// TIA Portal V20 export
FUNCTION_BLOCK "LSicar_KistlerPress"   // FB2, LAD
{ S7_Optimized_Access := 'TRUE' }
VERSION : 0.1
// stored: AutoNumber true, IsIECCheckEnabled false, IsRetainMemResEnabled false, MemoryReserve 100, SetENOAutomatically false, UDAEnableTagReadback false
   VAR_INPUT
      plantidentifier { ExternalAccessible := 'False'; ExternalVisible := 'False'; ExternalWritable := 'False'} : WString[24];
      CarrierID { ExternalAccessible := 'False'; ExternalVisible := 'False'; ExternalWritable := 'False'} : WString[9];
      mpSerialNumber { ExternalAccessible := 'False'; ExternalVisible := 'False'; ExternalWritable := 'False'} : String[24];
      additionaAlarmText { ExternalAccessible := 'False'; ExternalVisible := 'False'; ExternalWritable := 'False'} : WString[15];
      tecUnitNumber { ExternalAccessible := 'False'; ExternalVisible := 'False'; ExternalWritable := 'False'} : Int;
      enableBlock { ExternalAccessible := 'False'; ExternalVisible := 'False'; ExternalWritable := 'False'} : Bool := TRUE;
      HardwareOK { ExternalAccessible := 'False'; ExternalVisible := 'False'; ExternalWritable := 'False'} : Bool := TRUE;
      SafetyOK { ExternalAccessible := 'False'; ExternalVisible := 'False'; ExternalWritable := 'False'} : Bool := TRUE;
      servoNotInstalled { ExternalAccessible := 'False'; ExternalVisible := 'False'; ExternalWritable := 'False'} : Bool;
      hardwareID1 { ExternalAccessible := 'False'; ExternalVisible := 'False'; ExternalWritable := 'False'} : HW_IO;
      hardwareID2 { ExternalAccessible := 'False'; ExternalVisible := 'False'; ExternalWritable := 'False'} : HW_IO;
      smartClientIPAddress { ExternalAccessible := 'False'; ExternalVisible := 'False'; ExternalWritable := 'False'} : String[20];
      mpNumber { ExternalAccessible := 'False'; ExternalVisible := 'False'; ExternalWritable := 'False'} : Byte;
      cfgAdd { ExternalAccessible := 'False'; ExternalVisible := 'False'; ExternalWritable := 'False'} : Byte;
      CfgLentgh { ExternalAccessible := 'False'; ExternalVisible := 'False'; ExternalWritable := 'False'} : Byte;
      SelectPageNumber { ExternalAccessible := 'False'; ExternalVisible := 'False'; ExternalWritable := 'False'} : Byte;
      selectSequence { ExternalAccessible := 'False'; ExternalVisible := 'False'; ExternalWritable := 'False'} : Byte;
      extStopRequest { ExternalAccessible := 'False'; ExternalVisible := 'False'; ExternalWritable := 'False'} : Bool;
      strobeEnable { ExternalAccessible := 'False'; ExternalVisible := 'False'; ExternalWritable := 'False'} : Bool;
      startTL { ExternalAccessible := 'False'; ExternalVisible := 'False'; ExternalWritable := 'False'} : Bool;
      autoRunSequence { ExternalAccessible := 'False'; ExternalVisible := 'False'; ExternalWritable := 'False'} : Bool := FALSE;
      autoHomePosition { ExternalAccessible := 'False'; ExternalVisible := 'False'; ExternalWritable := 'False'} : Bool;
      autoDriveToReferencePosition { ExternalAccessible := 'False'; ExternalVisible := 'False'; ExternalWritable := 'False'} : Bool;
      JogFwd { ExternalAccessible := 'False'; ExternalVisible := 'False'; ExternalWritable := 'False'} : Bool;
      JogNeq { ExternalAccessible := 'False'; ExternalVisible := 'False'; ExternalWritable := 'False'} : Bool;
      continuewait { ExternalAccessible := 'False'; ExternalVisible := 'False'; ExternalWritable := 'False'} : Bool;
      SequenceEndReset { ExternalAccessible := 'False'; ExternalVisible := 'False'; ExternalWritable := 'False'} : Bool;
      enableRunSequence { ExternalAccessible := 'False'; ExternalVisible := 'False'; ExternalWritable := 'False'} : Bool := TRUE;
      enablehomePos { ExternalAccessible := 'False'; ExternalVisible := 'False'; ExternalWritable := 'False'} : Bool := TRUE;
      externalAlarm { ExternalAccessible := 'False'; ExternalVisible := 'False'; ExternalWritable := 'False'} : Bool;
      runWithoutEnable { ExternalAccessible := 'False'; ExternalVisible := 'False'; ExternalWritable := 'False'} : Bool;
      hideAlarmAll { ExternalAccessible := 'False'; ExternalVisible := 'False'; ExternalWritable := 'False'} : Bool;
      hideAlarmMask { ExternalAccessible := 'False'; ExternalVisible := 'False'; ExternalWritable := 'False'} : DWord;
      OpModeUserInterfaceOut { ExternalAccessible := 'False'; ExternalVisible := 'False'; ExternalWritable := 'False'} : "LSicar_typeOpmodeOut";
      timeOperation { ExternalAccessible := 'False'; ExternalVisible := 'False'; ExternalWritable := 'False'} : Time;
      timeExtStop { ExternalAccessible := 'False'; ExternalVisible := 'False'; ExternalWritable := 'False'} : Time;
      parameters { ExternalAccessible := 'False'; ExternalVisible := 'False'; ExternalWritable := 'False'} : "LDrive_typeKistlerParameters";
   END_VAR
   VAR_OUTPUT
      GeneralAlarm { ExternalAccessible := 'False'; ExternalVisible := 'False'; ExternalWritable := 'False'} : Bool;
      AutomaticActive { ExternalAccessible := 'False'; ExternalVisible := 'False'; ExternalWritable := 'False'} : Bool;
      okTotal { ExternalAccessible := 'False'; ExternalVisible := 'False'; ExternalWritable := 'False'} : Bool;
      nokTotal { ExternalAccessible := 'False'; ExternalVisible := 'False'; ExternalWritable := 'False'} : Bool;
      noPass { ExternalAccessible := 'False'; ExternalVisible := 'False'; ExternalWritable := 'False'} : Bool;
      sequenceRunning { ExternalAccessible := 'False'; ExternalVisible := 'False'; ExternalWritable := 'False'} : Bool;
      sequenceStopped { ExternalAccessible := 'False'; ExternalVisible := 'False'; ExternalWritable := 'False'} : Bool;
      Sequenceend { ExternalAccessible := 'False'; ExternalVisible := 'False'; ExternalWritable := 'False'} : Bool;
      homePos { ExternalAccessible := 'False'; ExternalVisible := 'False'; ExternalWritable := 'False'} : Bool;
      referencePos { ExternalAccessible := 'False'; ExternalVisible := 'False'; ExternalWritable := 'False'} : Bool;
      waitContinue { ExternalAccessible := 'False'; ExternalVisible := 'False'; ExternalWritable := 'False'} : Bool;
      ready { ExternalAccessible := 'False'; ExternalVisible := 'False'; ExternalWritable := 'False'} : Bool;
      pvCurrentValueX { ExternalAccessible := 'False'; ExternalVisible := 'False'; ExternalWritable := 'False'} : Real;
      pvCurrentValueY { ExternalAccessible := 'False'; ExternalVisible := 'False'; ExternalWritable := 'False'} : Real;
      pvCurveXminX { ExternalAccessible := 'False'; ExternalVisible := 'False'; ExternalWritable := 'False'} : Real;
      pvCurveXmaxX { ExternalAccessible := 'False'; ExternalVisible := 'False'; ExternalWritable := 'False'} : Real;
      pvCurveYminY { ExternalAccessible := 'False'; ExternalVisible := 'False'; ExternalWritable := 'False'} : Real;
      pvCurveYmaxY { ExternalAccessible := 'False'; ExternalVisible := 'False'; ExternalWritable := 'False'} : Real;
      customeProcessValues { ExternalAccessible := 'False'; ExternalVisible := 'False'; ExternalWritable := 'False'} : "LDrive_typeKistlerProcessValues";
      displayeservoJogSpeed { ExternalAccessible := 'False'; ExternalVisible := 'False'; ExternalWritable := 'False'} : Real;
      standstill { ExternalAccessible := 'False'; ExternalVisible := 'False'; ExternalWritable := 'False'} : Bool;
      MeasurementProgramEcho { ExternalAccessible := 'False'; ExternalVisible := 'False'; ExternalWritable := 'False'} : DInt;
      currentLabel { ExternalAccessible := 'False'; ExternalVisible := 'False'; ExternalWritable := 'False'} : Byte;
   END_VAR
   VAR_IN_OUT
      interfaceHmi : Array[*] of "LDrive_typeKistlerHmi";
   END_VAR
   VAR
      statDataExchangeReceive { ExternalAccessible := 'False'; ExternalVisible := 'False'; ExternalWritable := 'False'} : "LDrive_typeKistlerPressDataRecv";
      statDataExchangeSend { ExternalAccessible := 'False'; ExternalVisible := 'False'; ExternalWritable := 'False'} : "LDrive_typeKistlerPressDataSend";
      statInstruction { ExternalAccessible := 'False'; ExternalVisible := 'False'; ExternalWritable := 'False'} : Struct
         timeroperation { ExternalAccessible := 'False'; ExternalVisible := 'False'; ExternalWritable := 'False'; S7_SetPoint := 'True'} : IEC_TIMER;
         driveEnableTMR { ExternalAccessible := 'False'; ExternalVisible := 'False'; ExternalWritable := 'False'; S7_SetPoint := 'True'} : IEC_TIMER;
      END_STRUCT;
      stateAlarm { ExternalAccessible := 'False'; ExternalVisible := 'False'; ExternalWritable := 'False'} : Struct
         spare0 { ExternalAccessible := 'False'; ExternalVisible := 'False'; ExternalWritable := 'False'} : Bool;
         hardwareNOK { ExternalAccessible := 'False'; ExternalVisible := 'False'; ExternalWritable := 'False'} : Bool;
         driveenabledNOK { ExternalAccessible := 'False'; ExternalVisible := 'False'; ExternalWritable := 'False'} : Bool;
         enableRunSequence { ExternalAccessible := 'False'; ExternalVisible := 'False'; ExternalWritable := 'False'} : Bool;
         enableHomePos { ExternalAccessible := 'False'; ExternalVisible := 'False'; ExternalWritable := 'False'} : Bool;
         timerMonitorRunSequence { ExternalAccessible := 'False'; ExternalVisible := 'False'; ExternalWritable := 'False'} : Bool;
         timerMonitorHomePos { ExternalAccessible := 'False'; ExternalVisible := 'False'; ExternalWritable := 'False'} : Bool;
         timerMonitorReferencePos { ExternalAccessible := 'False'; ExternalVisible := 'False'; ExternalWritable := 'False'} : Bool;
         noContinueWaitCommand { ExternalAccessible := 'False'; ExternalVisible := 'False'; ExternalWritable := 'False'} : Bool;
         alarm { ExternalAccessible := 'False'; ExternalVisible := 'False'; ExternalWritable := 'False'} : Bool;
         spare11 { ExternalAccessible := 'False'; ExternalVisible := 'False'; ExternalWritable := 'False'} : Bool;
         smesActive { ExternalAccessible := 'False'; ExternalVisible := 'False'; ExternalWritable := 'False'} : Bool;
         safetyNOK { ExternalAccessible := 'False'; ExternalVisible := 'False'; ExternalWritable := 'False'} : Bool;
         smst2active { ExternalAccessible := 'False'; ExternalVisible := 'False'; ExternalWritable := 'False'} : Bool;
         smm1active { ExternalAccessible := 'False'; ExternalVisible := 'False'; ExternalWritable := 'False'} : Bool;
         serialnumbermismatch { ExternalAccessible := 'False'; ExternalVisible := 'False'; ExternalWritable := 'False'} : Bool;
         transmissionFault { ExternalAccessible := 'False'; ExternalVisible := 'False'; ExternalWritable := 'False'} : Bool;
         remoteControlNotActive { ExternalAccessible := 'False'; ExternalVisible := 'False'; ExternalWritable := 'False'} : Bool;
      END_STRUCT;
      stateHideAlarm { ExternalAccessible := 'False'; ExternalVisible := 'False'; ExternalWritable := 'False'} : Struct
         spare0 { ExternalAccessible := 'False'; ExternalVisible := 'False'; ExternalWritable := 'False'} : Bool;
         hardwareNOK { ExternalAccessible := 'False'; ExternalVisible := 'False'; ExternalWritable := 'False'} : Bool;
         transmissionFault { ExternalAccessible := 'False'; ExternalVisible := 'False'; ExternalWritable := 'False'} : Bool;
         driveEnabledNOK { ExternalAccessible := 'False'; ExternalVisible := 'False'; ExternalWritable := 'False'} : Bool;
         enableRunSequence { ExternalAccessible := 'False'; ExternalVisible := 'False'; ExternalWritable := 'False'} : Bool;
         enableHomePos { ExternalAccessible := 'False'; ExternalVisible := 'False'; ExternalWritable := 'False'} : Bool;
         timerMonitorRunSequence { ExternalAccessible := 'False'; ExternalVisible := 'False'; ExternalWritable := 'False'} : Bool;
         timerMonitorHomePos { ExternalAccessible := 'False'; ExternalVisible := 'False'; ExternalWritable := 'False'} : Bool;
         timerMonitorReferencePos { ExternalAccessible := 'False'; ExternalVisible := 'False'; ExternalWritable := 'False'} : Bool;
         noContinueWaitCommand { ExternalAccessible := 'False'; ExternalVisible := 'False'; ExternalWritable := 'False'} : Bool;
         Alarm { ExternalAccessible := 'False'; ExternalVisible := 'False'; ExternalWritable := 'False'} : Bool;
         spare11 { ExternalAccessible := 'False'; ExternalVisible := 'False'; ExternalWritable := 'False'} : Bool;
         smesactive { ExternalAccessible := 'False'; ExternalVisible := 'False'; ExternalWritable := 'False'} : Bool;
         safetyNOK { ExternalAccessible := 'False'; ExternalVisible := 'False'; ExternalWritable := 'False'} : Bool;
         smst2active { ExternalAccessible := 'False'; ExternalVisible := 'False'; ExternalWritable := 'False'} : Bool;
         smm1Active { ExternalAccessible := 'False'; ExternalVisible := 'False'; ExternalWritable := 'False'} : Bool;
      END_STRUCT;
      aux { ExternalAccessible := 'False'; ExternalVisible := 'False'; ExternalWritable := 'False'} : Struct
         generalAlarm { ExternalAccessible := 'False'; ExternalVisible := 'False'; ExternalWritable := 'False'} : Bool := false;
         plantIdentifier { ExternalAccessible := 'False'; ExternalVisible := 'False'; ExternalWritable := 'False'} : String[24];
         HideAlarmAll { ExternalAccessible := 'False'; ExternalVisible := 'False'; ExternalWritable := 'False'} : Bool := false;
         manualMode { ExternalAccessible := 'False'; ExternalVisible := 'False'; ExternalWritable := 'False'} : Bool := false;
         automaticMode { ExternalAccessible := 'False'; ExternalVisible := 'False'; ExternalWritable := 'False'} : Bool := false;
         singleStepMode { ExternalAccessible := 'False'; ExternalVisible := 'False'; ExternalWritable := 'False'} : Bool := false;
         setupMode { ExternalAccessible := 'False'; ExternalVisible := 'False'; ExternalWritable := 'False'} : Bool := false;
         externalAlarm { ExternalAccessible := 'False'; ExternalVisible := 'False'; ExternalWritable := 'False'} : Bool := false;
         alarmPdNoChange { ExternalAccessible := 'False'; ExternalVisible := 'False'; ExternalWritable := 'False'} : Bool := false;
         internalAlarmPdNoChange { ExternalAccessible := 'False'; ExternalVisible := 'False'; ExternalWritable := 'False'} : Bool := false;
         lastAlarmNoPD { ExternalAccessible := 'False'; ExternalVisible := 'False'; ExternalWritable := 'False'} : UInt := 0;
         lastInternalAlarmNoPD { ExternalAccessible := 'False'; ExternalVisible := 'False'; ExternalWritable := 'False'} : UInt := 0;
         enableAdvancedCodeView { ExternalAccessible := 'False'; ExternalVisible := 'False'; ExternalWritable := 'False'} : Bool := false;
         enableReverseCodeView { ExternalAccessible := 'False'; ExternalVisible := 'False'; ExternalWritable := 'False'} : Bool := false;
         codeViewAdvancedFilter { ExternalAccessible := 'False'; ExternalVisible := 'False'; ExternalWritable := 'False'} : WString[48];
         codeViewReverseFilter { ExternalAccessible := 'False'; ExternalVisible := 'False'; ExternalWritable := 'False'} : WString[48];
         iecTimer1 { ExternalAccessible := 'False'; ExternalVisible := 'False'; ExternalWritable := 'False'} : TON_TIME;
         logicEnable { ExternalAccessible := 'False'; ExternalVisible := 'False'; ExternalWritable := 'False'; S7_SetPoint := 'True'} : Bool := false;
         runSequence { ExternalAccessible := 'False'; ExternalVisible := 'False'; ExternalWritable := 'False'} : Bool := false;
         sequenceEnd { ExternalAccessible := 'False'; ExternalVisible := 'False'; ExternalWritable := 'False'} : Bool := false;
         dataStrobed { ExternalAccessible := 'False'; ExternalVisible := 'False'; ExternalWritable := 'False'} : Bool := false;
         SeqEnd { ExternalAccessible := 'False'; ExternalVisible := 'False'; ExternalWritable := 'False'} : Bool := false;
         remoteControl { ExternalAccessible := 'False'; ExternalVisible := 'False'; ExternalWritable := 'False'} : Bool := false;
         manualDataStrobe { ExternalAccessible := 'False'; ExternalVisible := 'False'; ExternalWritable := 'False'} : Bool := false;
         kistlerDataDB { ExternalAccessible := 'False'; ExternalVisible := 'False'; ExternalWritable := 'False'} : Int := 0;
         pulse { ExternalAccessible := 'False'; ExternalVisible := 'False'; ExternalWritable := 'False'} : Array[0..16] of Bool;
         Interface { ExternalAccessible := 'False'; ExternalVisible := 'False'; ExternalWritable := 'False'} : DWord;
      END_STRUCT;
      ons { ExternalAccessible := 'False'; ExternalVisible := 'False'; ExternalWritable := 'False'} : Array[0..16] of Bool;
      statTimeExpire { ExternalAccessible := 'False'; ExternalVisible := 'False'; ExternalWritable := 'False'} : Struct
         operating { ExternalAccessible := 'False'; ExternalVisible := 'False'; ExternalWritable := 'False'} : Bool;
         position_pLeft { ExternalAccessible := 'False'; ExternalVisible := 'False'; ExternalWritable := 'False'} : Bool;
         selaypair_mon { ExternalAccessible := 'False'; ExternalVisible := 'False'; ExternalWritable := 'False'} : Bool;
         dwellTimeWork { ExternalAccessible := 'False'; ExternalVisible := 'False'; ExternalWritable := 'False'} : Bool;
         dwellTimeHome { ExternalAccessible := 'False'; ExternalVisible := 'False'; ExternalWritable := 'False'} : Bool;
      END_STRUCT;
      statAlarmtextHeader { ExternalAccessible := 'False'; ExternalVisible := 'False'; ExternalWritable := 'False'} : WString[60];
      statAlarmtextFooter { ExternalAccessible := 'False'; ExternalVisible := 'False'; ExternalWritable := 'False'} : WString[24];
      statPalletID { ExternalAccessible := 'False'; ExternalVisible := 'False'; ExternalWritable := 'False'} : WString[9];
      statAlarmNoPD { ExternalAccessible := 'False'; ExternalVisible := 'False'; ExternalWritable := 'False'} : UInt;
      statInternalAlarmNoPD { ExternalAccessible := 'False'; ExternalVisible := 'False'; ExternalWritable := 'False'} : UInt;
      statHideAlarmMessagesPD { ExternalAccessible := 'False'; ExternalVisible := 'False'; ExternalWritable := 'False'} : Bool;
      statGlobalTecunitWarningTestListItem { ExternalAccessible := 'False'; ExternalVisible := 'False'; ExternalWritable := 'False'} : USInt := 92;
      statCodeViewAdvanceCond { ExternalAccessible := 'False'; ExternalVisible := 'False'; ExternalWritable := 'False'} : TON_TIME;
      statCodeViewReverseCond { ExternalAccessible := 'False'; ExternalVisible := 'False'; ExternalWritable := 'False'; S7_SetPoint := 'True'} : TON_TIME;
      statdriveDelayTimer { ExternalAccessible := 'False'; ExternalVisible := 'False'; ExternalWritable := 'False'; S7_SetPoint := 'True'} : TON_TIME;
      tof { ExternalAccessible := 'False'; ExternalVisible := 'False'; ExternalWritable := 'False'; S7_SetPoint := 'True'} : TON_TIME;
      statSerialByteIndex { ExternalAccessible := 'False'; ExternalVisible := 'False'; ExternalWritable := 'False'; S7_SetPoint := 'True'} : Int;
      statAlarmByteIndex { ExternalAccessible := 'False'; ExternalVisible := 'False'; ExternalWritable := 'False'} : Int;
      statStringIndex { ExternalAccessible := 'False'; ExternalVisible := 'False'; ExternalWritable := 'False'} : Int;
      statSerialOutput { ExternalAccessible := 'False'; ExternalVisible := 'False'; ExternalWritable := 'False'} : String[24];
      instKistlerOnDelay { ExternalAccessible := 'False'; ExternalVisible := 'False'; ExternalWritable := 'False'} : TON_TIME;
      internalFaultCode { ExternalAccessible := 'False'; ExternalVisible := 'False'; ExternalWritable := 'False'; S7_SetPoint := 'True'} : Array[0..63] of Bool;
      AlarmTextConstants { ExternalAccessible := 'False'; ExternalVisible := 'False'; ExternalWritable := 'False'} : Array[0..63] of Int;
      i { ExternalAccessible := 'False'; ExternalVisible := 'False'; ExternalWritable := 'False'} : Int;
   END_VAR
   VAR_TEMP
      tempReturnValueRead : Int;
      tempReturnValueWrite : Int;
      tempMPEcho : SInt;
      tempReadOK : Bool;
      tempWriteOK : Bool;
      tempValue : DWord;
      tempString : String[24];
      tempSerialLength : USInt;
      tempIndex : USInt;
      tempDword : DWord;
      tempErrorValue : Int;
      tempDint : DInt;
   END_VAR
   VAR CONSTANT
      cfgKistlerOnDelay : Time := T#1s;
   END_VAR
   VAR_TEMP   // added for the SCL form of the ladder/FBD networks
      _w1 : Bool;
      _w2 : Bool;
      _w3 : Bool;
      _w4 : Bool;
      _w5 : Bool;
      _w6 : Bool;
      _w7 : Bool;
   END_VAR
BEGIN

REGION Network 1 (SCL): Read RAW Data from Kistler
       #tempReturnValueRead := DPRD_DAT(LADDR := #hardwareID1, RECORD => #statDataExchangeReceive);    // Read from Kistler
END_REGION

REGION Network 2: Read OK
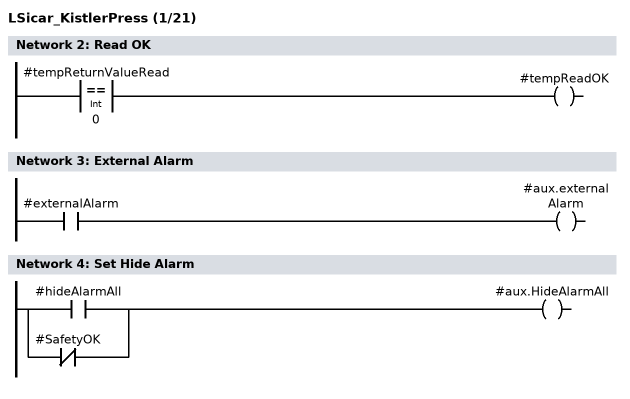
   RUNG wire#powerrail
      { S7_Templates := "SrcType := Int" } EQ_Contact(in1 := #tempReturnValueRead, in2 := 0)
      Coil( #tempReadOK )
   END_RUNG
   // the same network as SCL:
   #tempReadOK := #tempReturnValueRead = 0;
END_REGION

REGION Network 3: External Alarm
   RUNG wire#powerrail
      Contact( #externalAlarm )
      Coil( #aux.externalAlarm )
   END_RUNG
   // the same network as SCL:
   #aux.externalAlarm := #externalAlarm;
END_REGION

REGION Network 4: Set Hide Alarm
   RUNG wire#powerrail
      Contact( #hideAlarmAll )
      wire#w1
      Coil( #aux.HideAlarmAll )
   END_RUNG
   RUNG wire#powerrail
      I_Contact( #SafetyOK )
   END_RUNG wire#w1
   // the same network as SCL:
   #aux.HideAlarmAll := #hideAlarmAll OR NOT #SafetyOK;
END_REGION

REGION Network 5: Hide Alarm
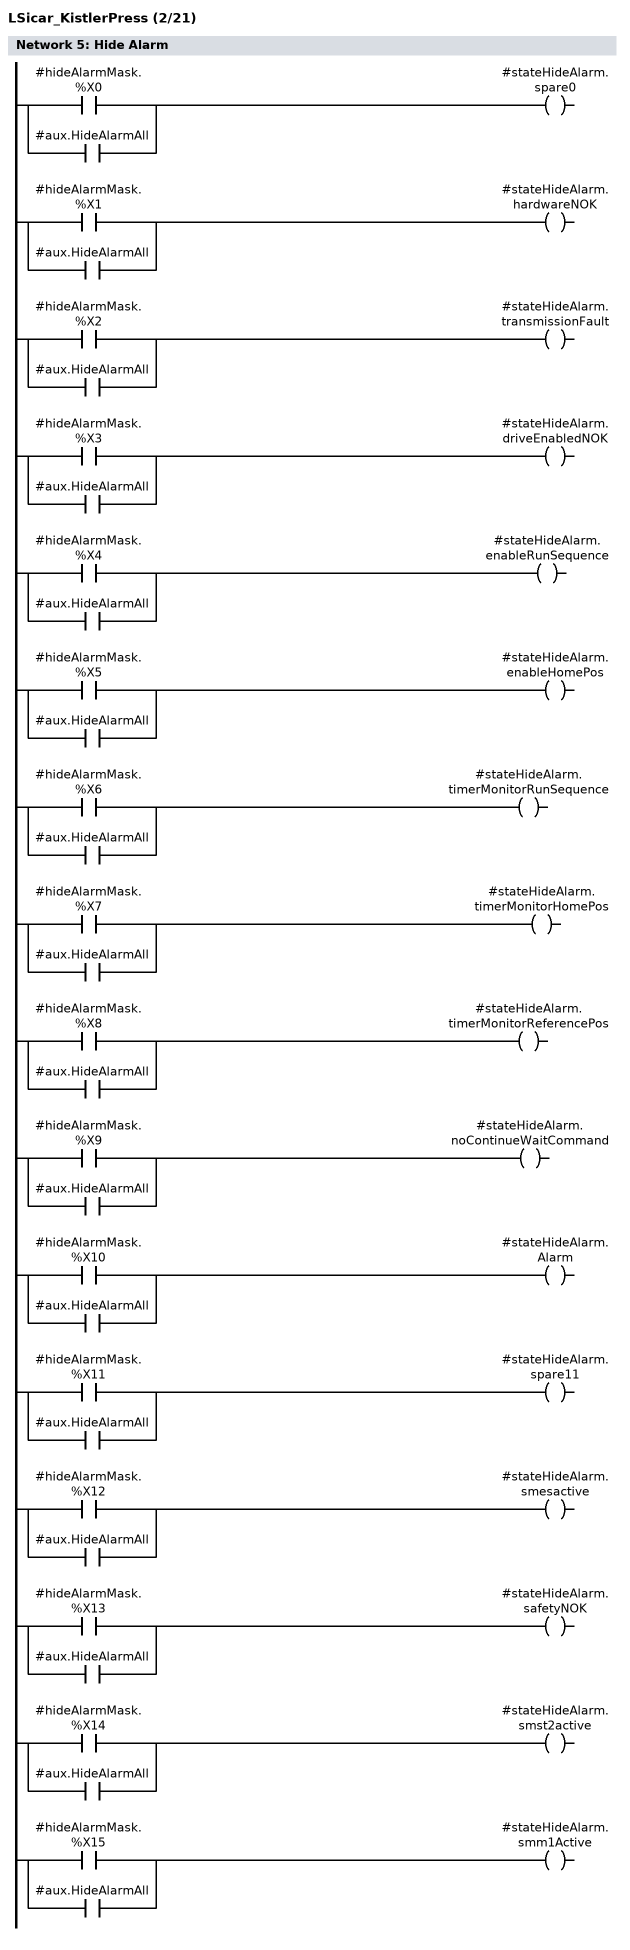
   RUNG wire#powerrail
      Contact( #hideAlarmMask.%X0 )
      wire#w1
      Coil( #stateHideAlarm.spare0 )
   END_RUNG
   RUNG wire#powerrail
      Contact( #aux.HideAlarmAll )
   END_RUNG wire#w1
   RUNG wire#powerrail
      Contact( #hideAlarmMask.%X1 )
      wire#w2
      Coil( #stateHideAlarm.hardwareNOK )
   END_RUNG
   RUNG wire#powerrail
      Contact( #aux.HideAlarmAll )
   END_RUNG wire#w2
   RUNG wire#powerrail
      Contact( #hideAlarmMask.%X2 )
      wire#w3
      Coil( #stateHideAlarm.transmissionFault )
   END_RUNG
   RUNG wire#powerrail
      Contact( #aux.HideAlarmAll )
   END_RUNG wire#w3
   RUNG wire#powerrail
      Contact( #hideAlarmMask.%X3 )
      wire#w4
      Coil( #stateHideAlarm.driveEnabledNOK )
   END_RUNG
   RUNG wire#powerrail
      Contact( #aux.HideAlarmAll )
   END_RUNG wire#w4
   RUNG wire#powerrail
      Contact( #hideAlarmMask.%X4 )
      wire#w5
      Coil( #stateHideAlarm.enableRunSequence )
   END_RUNG
   RUNG wire#powerrail
      Contact( #aux.HideAlarmAll )
   END_RUNG wire#w5
   RUNG wire#powerrail
      Contact( #hideAlarmMask.%X5 )
      wire#w6
      Coil( #stateHideAlarm.enableHomePos )
   END_RUNG
   RUNG wire#powerrail
      Contact( #aux.HideAlarmAll )
   END_RUNG wire#w6
   RUNG wire#powerrail
      Contact( #hideAlarmMask.%X6 )
      wire#w7
      Coil( #stateHideAlarm.timerMonitorRunSequence )
   END_RUNG
   RUNG wire#powerrail
      Contact( #aux.HideAlarmAll )
   END_RUNG wire#w7
   RUNG wire#powerrail
      Contact( #hideAlarmMask.%X7 )
      wire#w8
      Coil( #stateHideAlarm.timerMonitorHomePos )
   END_RUNG
   RUNG wire#powerrail
      Contact( #aux.HideAlarmAll )
   END_RUNG wire#w8
   RUNG wire#powerrail
      Contact( #hideAlarmMask.%X8 )
      wire#w9
      Coil( #stateHideAlarm.timerMonitorReferencePos )
   END_RUNG
   RUNG wire#powerrail
      Contact( #aux.HideAlarmAll )
   END_RUNG wire#w9
   RUNG wire#powerrail
      Contact( #hideAlarmMask.%X9 )
      wire#w10
      Coil( #stateHideAlarm.noContinueWaitCommand )
   END_RUNG
   RUNG wire#powerrail
      Contact( #aux.HideAlarmAll )
   END_RUNG wire#w10
   RUNG wire#powerrail
      Contact( #hideAlarmMask.%X10 )
      wire#w11
      Coil( #stateHideAlarm.Alarm )
   END_RUNG
   RUNG wire#powerrail
      Contact( #aux.HideAlarmAll )
   END_RUNG wire#w11
   RUNG wire#powerrail
      Contact( #hideAlarmMask.%X11 )
      wire#w12
      Coil( #stateHideAlarm.spare11 )
   END_RUNG
   RUNG wire#powerrail
      Contact( #aux.HideAlarmAll )
   END_RUNG wire#w12
   RUNG wire#powerrail
      Contact( #hideAlarmMask.%X12 )
      wire#w13
      Coil( #stateHideAlarm.smesactive )
   END_RUNG
   RUNG wire#powerrail
      Contact( #aux.HideAlarmAll )
   END_RUNG wire#w13
   RUNG wire#powerrail
      Contact( #hideAlarmMask.%X13 )
      wire#w14
      Coil( #stateHideAlarm.safetyNOK )
   END_RUNG
   RUNG wire#powerrail
      Contact( #aux.HideAlarmAll )
   END_RUNG wire#w14
   RUNG wire#powerrail
      Contact( #hideAlarmMask.%X14 )
      wire#w15
      Coil( #stateHideAlarm.smst2active )
   END_RUNG
   RUNG wire#powerrail
      Contact( #aux.HideAlarmAll )
   END_RUNG wire#w15
   RUNG wire#powerrail
      Contact( #hideAlarmMask.%X15 )
      wire#w16
      Coil( #stateHideAlarm.smm1Active )
   END_RUNG
   RUNG wire#powerrail
      Contact( #aux.HideAlarmAll )
   END_RUNG wire#w16
   // the same network as SCL:
   #stateHideAlarm.spare0 := #hideAlarmMask.%X0 OR #aux.HideAlarmAll;
   #stateHideAlarm.hardwareNOK := #hideAlarmMask.%X1 OR #aux.HideAlarmAll;
   #stateHideAlarm.transmissionFault := #hideAlarmMask.%X2 OR #aux.HideAlarmAll;
   #stateHideAlarm.driveEnabledNOK := #hideAlarmMask.%X3 OR #aux.HideAlarmAll;
   #stateHideAlarm.enableRunSequence := #hideAlarmMask.%X4 OR #aux.HideAlarmAll;
   #stateHideAlarm.enableHomePos := #hideAlarmMask.%X5 OR #aux.HideAlarmAll;
   #stateHideAlarm.timerMonitorRunSequence := #hideAlarmMask.%X6 OR #aux.HideAlarmAll;
   #stateHideAlarm.timerMonitorHomePos := #hideAlarmMask.%X7 OR #aux.HideAlarmAll;
   #stateHideAlarm.timerMonitorReferencePos := #hideAlarmMask.%X8 OR #aux.HideAlarmAll;
   #stateHideAlarm.noContinueWaitCommand := #hideAlarmMask.%X9 OR #aux.HideAlarmAll;
   #stateHideAlarm.Alarm := #hideAlarmMask.%X10 OR #aux.HideAlarmAll;
   #stateHideAlarm.spare11 := #hideAlarmMask.%X11 OR #aux.HideAlarmAll;
   #stateHideAlarm.smesactive := #hideAlarmMask.%X12 OR #aux.HideAlarmAll;
   #stateHideAlarm.safetyNOK := #hideAlarmMask.%X13 OR #aux.HideAlarmAll;
   #stateHideAlarm.smst2active := #hideAlarmMask.%X14 OR #aux.HideAlarmAll;
   #stateHideAlarm.smm1Active := #hideAlarmMask.%X15 OR #aux.HideAlarmAll;
END_REGION

REGION Network 6: Mode Selection
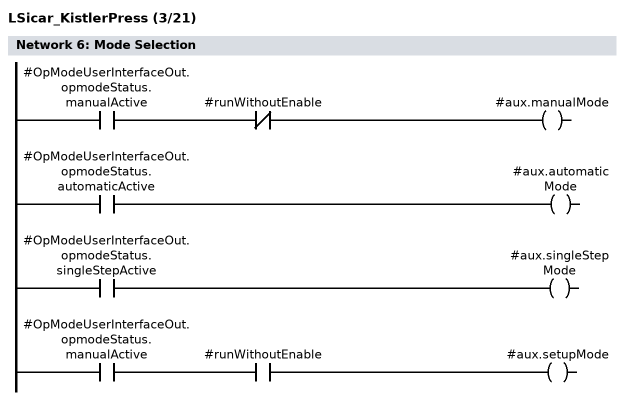
   RUNG wire#powerrail
      Contact( #OpModeUserInterfaceOut.opmodeStatus.manualActive )
      I_Contact( #runWithoutEnable )
      Coil( #aux.manualMode )
   END_RUNG
   RUNG wire#powerrail
      Contact( #OpModeUserInterfaceOut.opmodeStatus.automaticActive )
      Coil( #aux.automaticMode )
   END_RUNG
   RUNG wire#powerrail
      Contact( #OpModeUserInterfaceOut.opmodeStatus.singleStepActive )
      Coil( #aux.singleStepMode )
   END_RUNG
   RUNG wire#powerrail
      Contact( #OpModeUserInterfaceOut.opmodeStatus.manualActive )
      Contact( #runWithoutEnable )
      Coil( #aux.setupMode )
   END_RUNG
   // the same network as SCL:
   #aux.manualMode := #OpModeUserInterfaceOut.opmodeStatus.manualActive AND NOT #runWithoutEnable;
   #aux.automaticMode := #OpModeUserInterfaceOut.opmodeStatus.automaticActive;
   #aux.singleStepMode := #OpModeUserInterfaceOut.opmodeStatus.singleStepActive;
   #aux.setupMode := #OpModeUserInterfaceOut.opmodeStatus.manualActive AND #runWithoutEnable;
END_REGION

REGION Network 7: Clear Faults
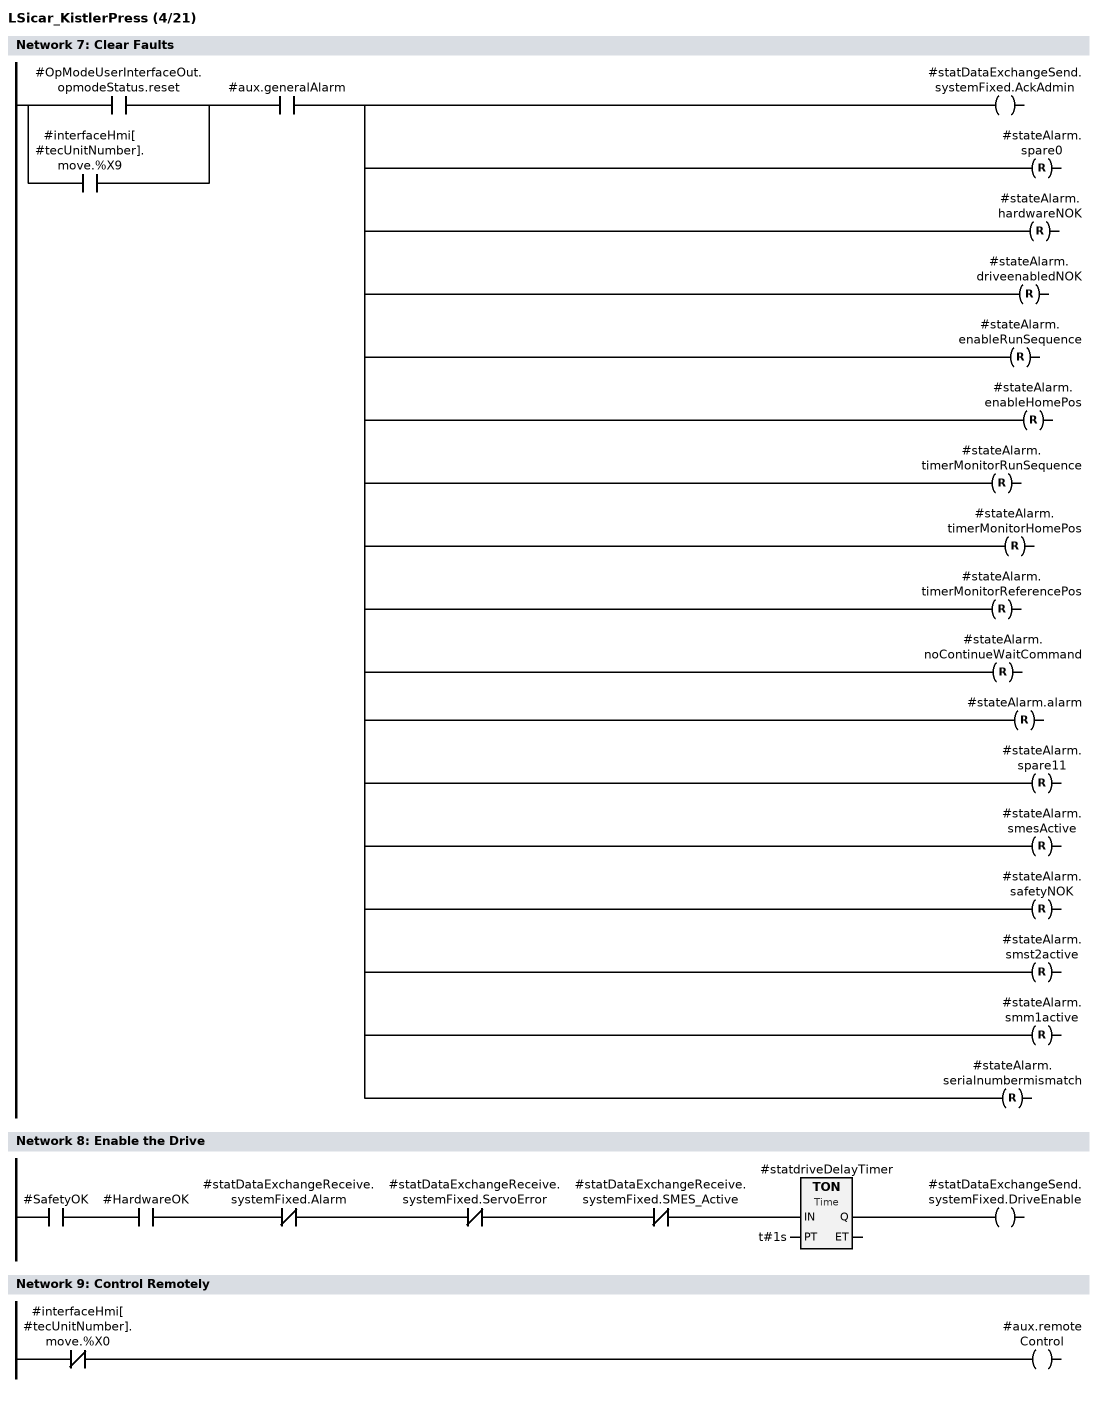
   RUNG wire#powerrail
      Contact( #OpModeUserInterfaceOut.opmodeStatus.reset )
      wire#w1
      Contact( #aux.generalAlarm )
      wire#w2
      Coil( #statDataExchangeSend.systemFixed.AckAdmin )
   END_RUNG
   RUNG wire#powerrail
      Contact( #interfaceHmi[#tecUnitNumber].move.%X9 )
   END_RUNG wire#w1
   RUNG wire#w2
      R_Coil( #stateAlarm.spare0 )
   END_RUNG
   RUNG wire#w2
      R_Coil( #stateAlarm.hardwareNOK )
   END_RUNG
   RUNG wire#w2
      R_Coil( #stateAlarm.driveenabledNOK )
   END_RUNG
   RUNG wire#w2
      R_Coil( #stateAlarm.enableRunSequence )
   END_RUNG
   RUNG wire#w2
      R_Coil( #stateAlarm.enableHomePos )
   END_RUNG
   RUNG wire#w2
      R_Coil( #stateAlarm.timerMonitorRunSequence )
   END_RUNG
   RUNG wire#w2
      R_Coil( #stateAlarm.timerMonitorHomePos )
   END_RUNG
   RUNG wire#w2
      R_Coil( #stateAlarm.timerMonitorReferencePos )
   END_RUNG
   RUNG wire#w2
      R_Coil( #stateAlarm.noContinueWaitCommand )
   END_RUNG
   RUNG wire#w2
      R_Coil( #stateAlarm.alarm )
   END_RUNG
   RUNG wire#w2
      R_Coil( #stateAlarm.spare11 )
   END_RUNG
   RUNG wire#w2
      R_Coil( #stateAlarm.smesActive )
   END_RUNG
   RUNG wire#w2
      R_Coil( #stateAlarm.safetyNOK )
   END_RUNG
   RUNG wire#w2
      R_Coil( #stateAlarm.smst2active )
   END_RUNG
   RUNG wire#w2
      R_Coil( #stateAlarm.smm1active )
   END_RUNG
   RUNG wire#w2
      R_Coil( #stateAlarm.serialnumbermismatch )
   END_RUNG
   // the same network as SCL:
   #statDataExchangeSend.systemFixed.AckAdmin := (#OpModeUserInterfaceOut.opmodeStatus.reset OR #interfaceHmi[#tecUnitNumber].move.%X9) AND #aux.generalAlarm;
   IF #statDataExchangeSend.systemFixed.AckAdmin THEN
       #stateAlarm.spare0 := FALSE;
       #stateAlarm.hardwareNOK := FALSE;
       #stateAlarm.driveenabledNOK := FALSE;
       #stateAlarm.enableRunSequence := FALSE;
       #stateAlarm.enableHomePos := FALSE;
       #stateAlarm.timerMonitorRunSequence := FALSE;
       #stateAlarm.timerMonitorHomePos := FALSE;
       #stateAlarm.timerMonitorReferencePos := FALSE;
       #stateAlarm.noContinueWaitCommand := FALSE;
       #stateAlarm.alarm := FALSE;
       #stateAlarm.spare11 := FALSE;
       #stateAlarm.smesActive := FALSE;
       #stateAlarm.safetyNOK := FALSE;
       #stateAlarm.smst2active := FALSE;
       #stateAlarm.smm1active := FALSE;
       #stateAlarm.serialnumbermismatch := FALSE;
   END_IF;
END_REGION

REGION Network 8: Enable the Drive
   RUNG wire#powerrail
      Contact( #SafetyOK )
      Contact( #HardwareOK )
      I_Contact( #statDataExchangeReceive.systemFixed.Alarm )
      I_Contact( #statDataExchangeReceive.systemFixed.ServoError )
      I_Contact( #statDataExchangeReceive.systemFixed.SMES_Active )
      { S7_Templates := "time_type := Time" } #statdriveDelayTimer.TON(pt := t#1s, et =>)
      Coil( #statDataExchangeSend.systemFixed.DriveEnable )
   END_RUNG
   // the same network as SCL:
   #statdriveDelayTimer(IN := #SafetyOK AND #HardwareOK AND NOT #statDataExchangeReceive.systemFixed.Alarm AND NOT #statDataExchangeReceive.systemFixed.ServoError AND NOT #statDataExchangeReceive.systemFixed.SMES_Active,   // TON
                        PT := t#1s);
   #statDataExchangeSend.systemFixed.DriveEnable := #statdriveDelayTimer.Q;
END_REGION

REGION Network 9: Control Remotely
   RUNG wire#powerrail
      I_Contact( #interfaceHmi[#tecUnitNumber].move.%X0 )
      Coil( #aux.remoteControl )
   END_RUNG
   // the same network as SCL:
   #aux.remoteControl := NOT #interfaceHmi[#tecUnitNumber].move.%X0;
END_REGION

REGION Network 10: Turn to Auto mode remotely
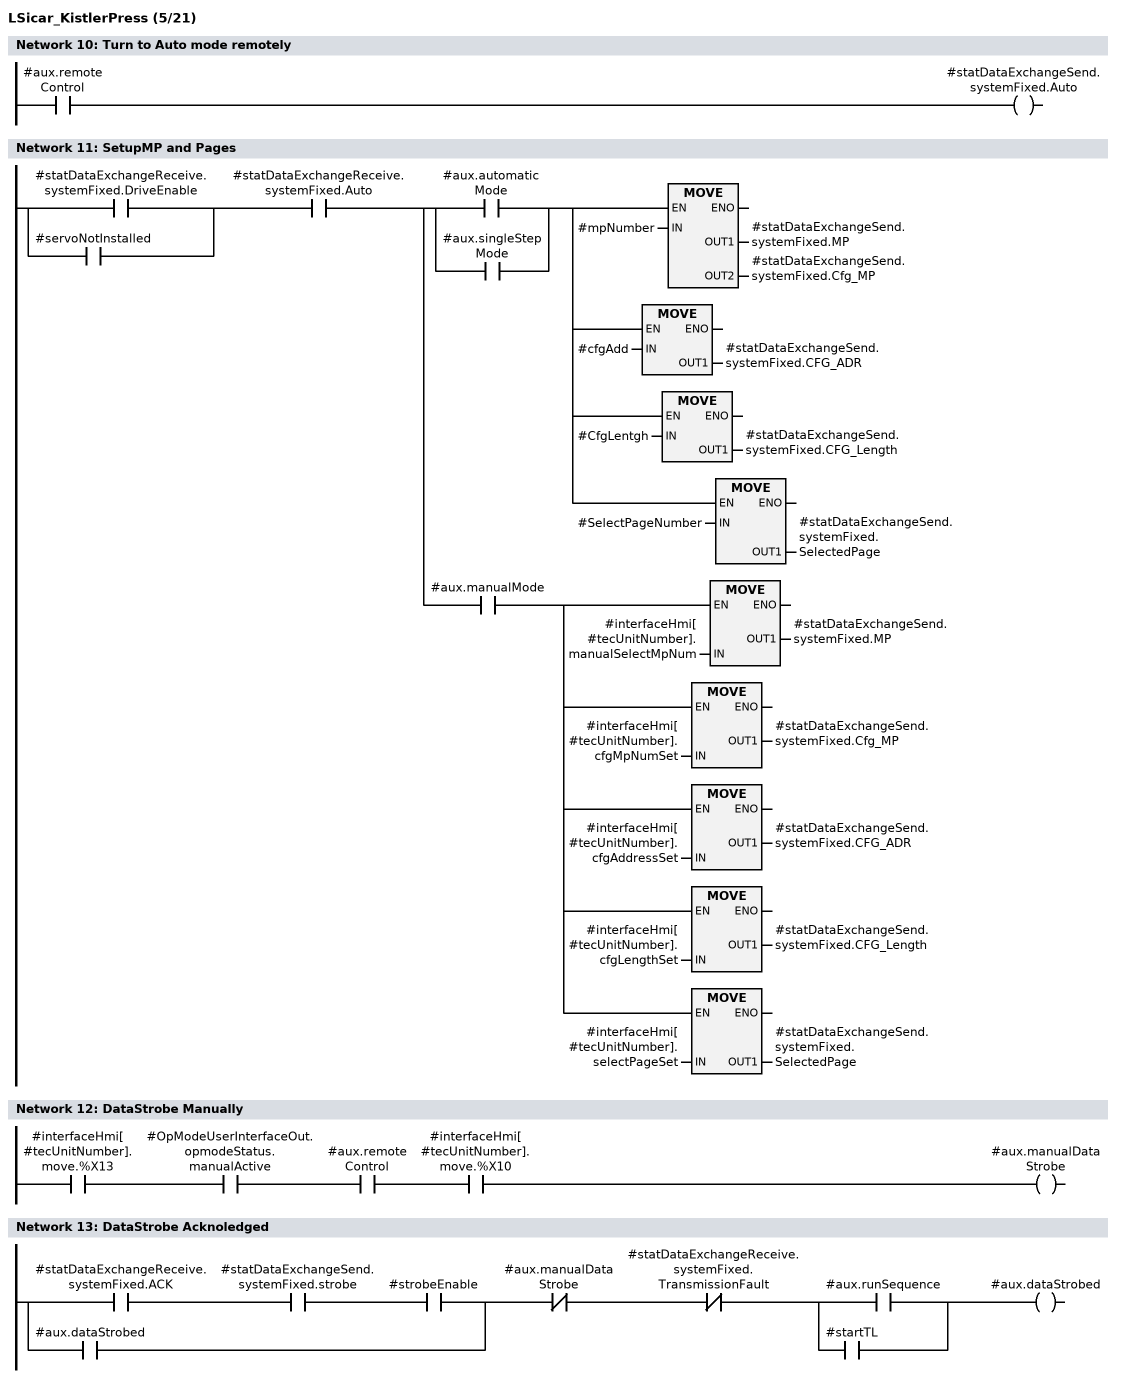
   RUNG wire#powerrail
      Contact( #aux.remoteControl )
      Coil( #statDataExchangeSend.systemFixed.Auto )
   END_RUNG
   // the same network as SCL:
   #statDataExchangeSend.systemFixed.Auto := #aux.remoteControl;
END_REGION

REGION Network 11: SetupMP and Pages
   RUNG wire#powerrail
      Contact( #statDataExchangeReceive.systemFixed.DriveEnable )
      wire#w1
      Contact( #statDataExchangeReceive.systemFixed.Auto )
      wire#w2
      Contact( #aux.automaticMode )
      wire#w3
      Move(in := #mpNumber, out1 => #statDataExchangeSend.systemFixed.MP, out2 => #statDataExchangeSend.systemFixed.Cfg_MP)
   END_RUNG
   RUNG wire#powerrail
      Contact( #servoNotInstalled )
   END_RUNG wire#w1
   RUNG wire#w2
      Contact( #aux.singleStepMode )
   END_RUNG wire#w3
   RUNG wire#w3
      Move(in := #cfgAdd, out1 => #statDataExchangeSend.systemFixed.CFG_ADR)
   END_RUNG
   RUNG wire#w3
      Move(in := #CfgLentgh, out1 => #statDataExchangeSend.systemFixed.CFG_Length)
   END_RUNG
   RUNG wire#w3
      Move(in := #SelectPageNumber, out1 => #statDataExchangeSend.systemFixed.SelectedPage)
   END_RUNG
   RUNG wire#w2
      Contact( #aux.manualMode )
      wire#w4
      Move(in := #interfaceHmi[#tecUnitNumber].manualSelectMpNum, out1 => #statDataExchangeSend.systemFixed.MP)
   END_RUNG
   RUNG wire#w4
      Move(in := #interfaceHmi[#tecUnitNumber].cfgMpNumSet, out1 => #statDataExchangeSend.systemFixed.Cfg_MP)
   END_RUNG
   RUNG wire#w4
      Move(in := #interfaceHmi[#tecUnitNumber].cfgAddressSet, out1 => #statDataExchangeSend.systemFixed.CFG_ADR)
   END_RUNG
   RUNG wire#w4
      Move(in := #interfaceHmi[#tecUnitNumber].cfgLengthSet, out1 => #statDataExchangeSend.systemFixed.CFG_Length)
   END_RUNG
   RUNG wire#w4
      Move(in := #interfaceHmi[#tecUnitNumber].selectPageSet, out1 => #statDataExchangeSend.systemFixed.SelectedPage)
   END_RUNG
   // the same network as SCL:
   #_w1 := (#statDataExchangeReceive.systemFixed.DriveEnable OR #servoNotInstalled) AND #statDataExchangeReceive.systemFixed.Auto;
   IF #_w1 AND (#aux.automaticMode OR #aux.singleStepMode) THEN
       #statDataExchangeSend.systemFixed.MP := #mpNumber;
       #statDataExchangeSend.systemFixed.Cfg_MP := #mpNumber;
       #statDataExchangeSend.systemFixed.CFG_ADR := #cfgAdd;
       #statDataExchangeSend.systemFixed.CFG_Length := #CfgLentgh;
       #statDataExchangeSend.systemFixed.SelectedPage := #SelectPageNumber;
   END_IF;
   IF #_w1 AND #aux.manualMode THEN
       #statDataExchangeSend.systemFixed.MP := #interfaceHmi[#tecUnitNumber].manualSelectMpNum;
       #statDataExchangeSend.systemFixed.Cfg_MP := #interfaceHmi[#tecUnitNumber].cfgMpNumSet;
       #statDataExchangeSend.systemFixed.CFG_ADR := #interfaceHmi[#tecUnitNumber].cfgAddressSet;
       #statDataExchangeSend.systemFixed.CFG_Length := #interfaceHmi[#tecUnitNumber].cfgLengthSet;
       #statDataExchangeSend.systemFixed.SelectedPage := #interfaceHmi[#tecUnitNumber].selectPageSet;
   END_IF;
END_REGION

REGION Network 12: DataStrobe Manually
   RUNG wire#powerrail
      Contact( #interfaceHmi[#tecUnitNumber].move.%X13 )
      Contact( #OpModeUserInterfaceOut.opmodeStatus.manualActive )
      Contact( #aux.remoteControl )
      Contact( #interfaceHmi[#tecUnitNumber].move.%X10 )
      Coil( #aux.manualDataStrobe )
   END_RUNG
   // the same network as SCL:
   #aux.manualDataStrobe := #interfaceHmi[#tecUnitNumber].move.%X13 AND #OpModeUserInterfaceOut.opmodeStatus.manualActive AND #aux.remoteControl AND #interfaceHmi[#tecUnitNumber].move.%X10;
END_REGION

REGION Network 13: DataStrobe Acknoledged
   RUNG wire#powerrail
      Contact( #statDataExchangeReceive.systemFixed.ACK )
      Contact( #statDataExchangeSend.systemFixed.strobe )
      Contact( #strobeEnable )
      wire#w1
      I_Contact( #aux.manualDataStrobe )
      I_Contact( #statDataExchangeReceive.systemFixed.TransmissionFault )
      wire#w2
      Contact( #aux.runSequence )
      wire#w3
      Coil( #aux.dataStrobed )
   END_RUNG
   RUNG wire#powerrail
      Contact( #aux.dataStrobed )
   END_RUNG wire#w1
   RUNG wire#w2
      Contact( #startTL )
   END_RUNG wire#w3
   // the same network as SCL:
   #aux.dataStrobed := ((#statDataExchangeReceive.systemFixed.ACK AND #statDataExchangeSend.systemFixed.strobe AND #strobeEnable) OR #aux.dataStrobed) AND NOT #aux.manualDataStrobe AND NOT #statDataExchangeReceive.systemFixed.TransmissionFault AND (#aux.runSequence OR #startTL);
END_REGION

REGION Network 14: Strobe data
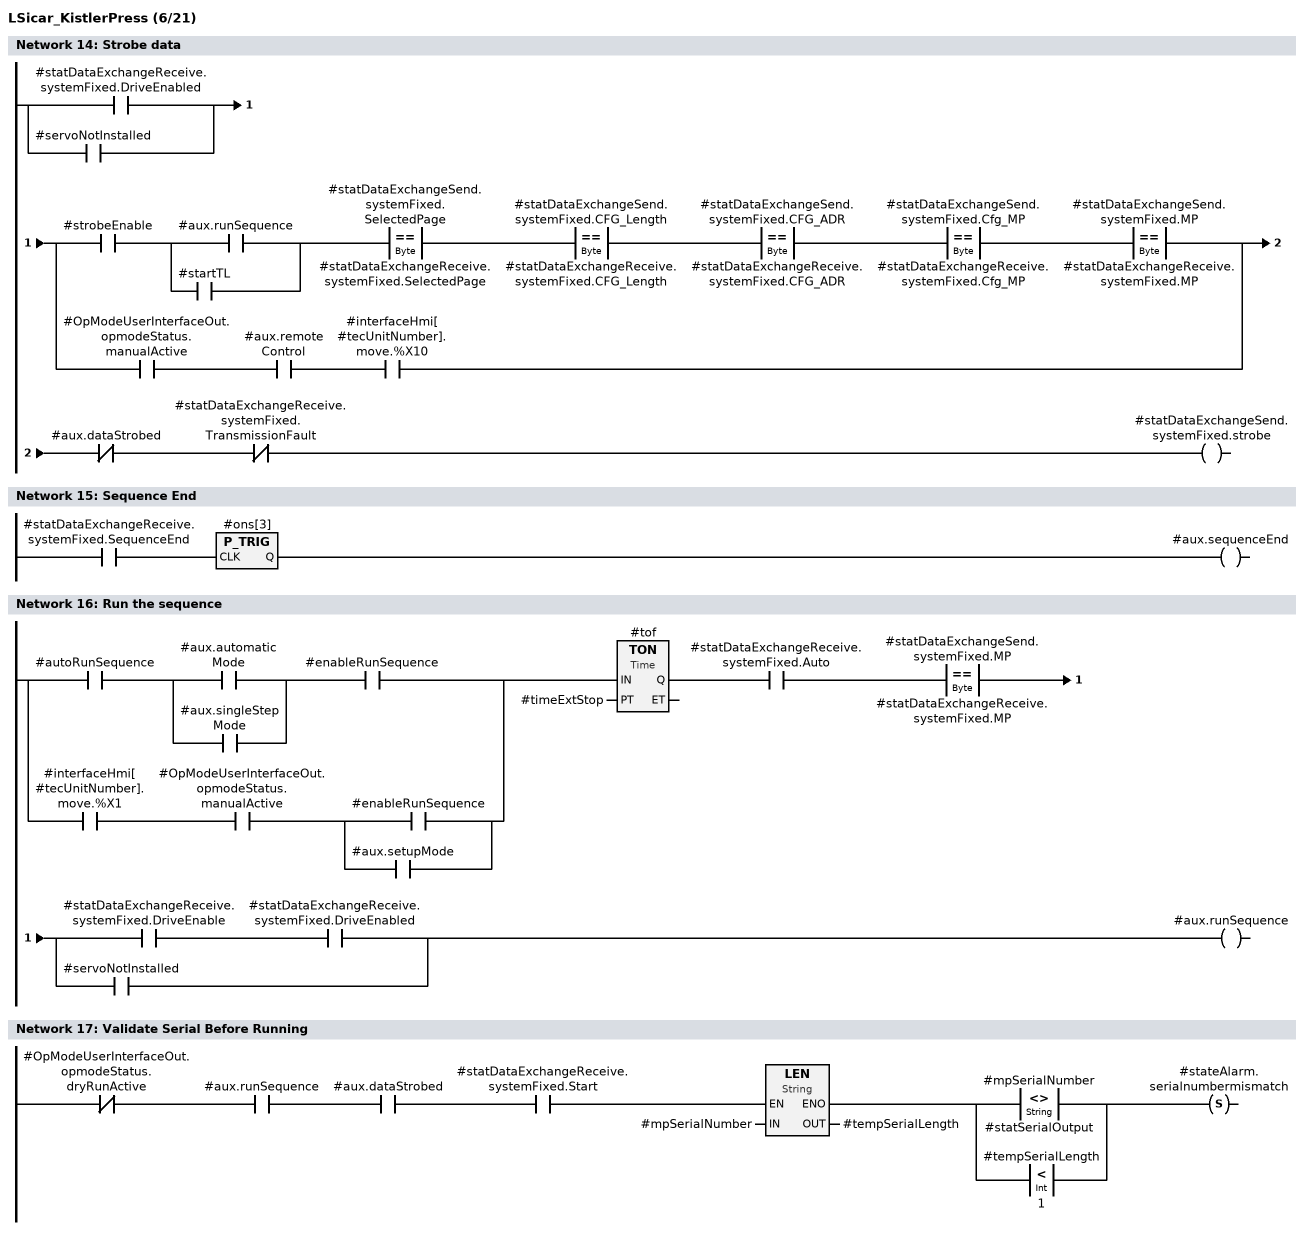
   RUNG wire#powerrail
      Contact( #statDataExchangeReceive.systemFixed.DriveEnabled )
      wire#w1
      Contact( #strobeEnable )
      wire#w2
      Contact( #aux.runSequence )
      wire#w3
      { S7_Templates := "SrcType := Byte" } EQ_Contact(in1 := #statDataExchangeSend.systemFixed.SelectedPage, in2 := #statDataExchangeReceive.systemFixed.SelectedPage)
      { S7_Templates := "SrcType := Byte" } EQ_Contact(in1 := #statDataExchangeSend.systemFixed.CFG_Length, in2 := #statDataExchangeReceive.systemFixed.CFG_Length)
      { S7_Templates := "SrcType := Byte" } EQ_Contact(in1 := #statDataExchangeSend.systemFixed.CFG_ADR, in2 := #statDataExchangeReceive.systemFixed.CFG_ADR)
      { S7_Templates := "SrcType := Byte" } EQ_Contact(in1 := #statDataExchangeSend.systemFixed.Cfg_MP, in2 := #statDataExchangeReceive.systemFixed.Cfg_MP)
      { S7_Templates := "SrcType := Byte" } EQ_Contact(in1 := #statDataExchangeSend.systemFixed.MP, in2 := #statDataExchangeReceive.systemFixed.MP)
      wire#w4
      I_Contact( #aux.dataStrobed )
      I_Contact( #statDataExchangeReceive.systemFixed.TransmissionFault )
      Coil( #statDataExchangeSend.systemFixed.strobe )
   END_RUNG
   RUNG wire#powerrail
      Contact( #servoNotInstalled )
   END_RUNG wire#w1
   RUNG wire#w2
      Contact( #startTL )
   END_RUNG wire#w3
   RUNG wire#w1
      Contact( #OpModeUserInterfaceOut.opmodeStatus.manualActive )
      Contact( #aux.remoteControl )
      Contact( #interfaceHmi[#tecUnitNumber].move.%X10 )
   END_RUNG wire#w4
   // the same network as SCL:
   #statDataExchangeSend.systemFixed.strobe := (#statDataExchangeReceive.systemFixed.DriveEnabled OR #servoNotInstalled) AND ((#strobeEnable AND (#aux.runSequence OR #startTL) AND (#statDataExchangeSend.systemFixed.SelectedPage = #statDataExchangeReceive.systemFixed.SelectedPage) AND (#statDataExchangeSend.systemFixed.CFG_Length = #statDataExchangeReceive.systemFixed.CFG_Length) AND (#statDataExchangeSend.systemFixed.CFG_ADR = #statDataExchangeReceive.systemFixed.CFG_ADR) AND (#statDataExchangeSend.systemFixed.Cfg_MP = #statDataExchangeReceive.systemFixed.Cfg_MP) AND (#statDataExchangeSend.systemFixed.MP = #statDataExchangeReceive.systemFixed.MP)) OR (#OpModeUserInterfaceOut.opmodeStatus.manualActive AND #aux.remoteControl AND #interfaceHmi[#tecUnitNumber].move.%X10)) AND NOT #aux.dataStrobed AND NOT #statDataExchangeReceive.systemFixed.TransmissionFault;
END_REGION

REGION Network 15: Sequence End
   RUNG wire#powerrail
      Contact( #statDataExchangeReceive.systemFixed.SequenceEnd )
      P_Trig( #ons[3] )
      Coil( #aux.sequenceEnd )
   END_RUNG
   // the same network as SCL:
   #_w1 := #statDataExchangeReceive.systemFixed.SequenceEnd AND NOT #ons[3];   // rising edge
   #ons[3] := #statDataExchangeReceive.systemFixed.SequenceEnd;
   #aux.sequenceEnd := #_w1;
END_REGION

REGION Network 16: Run the sequence
   RUNG wire#powerrail
      Contact( #autoRunSequence )
      wire#w1
      Contact( #aux.automaticMode )
      wire#w2
      Contact( #enableRunSequence )
      wire#w3
      { S7_Templates := "time_type := Time" } #tof.TON(pt := #timeExtStop, et =>)
      Contact( #statDataExchangeReceive.systemFixed.Auto )
      { S7_Templates := "SrcType := Byte" } EQ_Contact(in1 := #statDataExchangeSend.systemFixed.MP, in2 := #statDataExchangeReceive.systemFixed.MP)
      wire#w5
      Contact( #statDataExchangeReceive.systemFixed.DriveEnable )
      Contact( #statDataExchangeReceive.systemFixed.DriveEnabled )
      wire#w6
      Coil( #aux.runSequence )
   END_RUNG
   RUNG wire#w1
      Contact( #aux.singleStepMode )
   END_RUNG wire#w2
   RUNG wire#powerrail
      Contact( #interfaceHmi[#tecUnitNumber].move.%X1 )
      Contact( #OpModeUserInterfaceOut.opmodeStatus.manualActive )
      wire#w4
      Contact( #enableRunSequence )
   END_RUNG wire#w3
   RUNG wire#w4
      Contact( #aux.setupMode )
   END_RUNG wire#w3
   RUNG wire#w5
      Contact( #servoNotInstalled )
   END_RUNG wire#w6
   // the same network as SCL:
   #tof(IN := (#autoRunSequence AND (#aux.automaticMode OR #aux.singleStepMode) AND #enableRunSequence) OR (#interfaceHmi[#tecUnitNumber].move.%X1 AND #OpModeUserInterfaceOut.opmodeStatus.manualActive AND (#enableRunSequence OR #aux.setupMode)),   // TON
        PT := #timeExtStop);
   #aux.runSequence := #tof.Q AND #statDataExchangeReceive.systemFixed.Auto AND (#statDataExchangeSend.systemFixed.MP = #statDataExchangeReceive.systemFixed.MP) AND ((#statDataExchangeReceive.systemFixed.DriveEnable AND #statDataExchangeReceive.systemFixed.DriveEnabled) OR #servoNotInstalled);
END_REGION

REGION Network 17: Validate Serial Before Running
   RUNG wire#powerrail
      I_Contact( #OpModeUserInterfaceOut.opmodeStatus.dryRunActive )
      Contact( #aux.runSequence )
      Contact( #aux.dataStrobed )
      Contact( #statDataExchangeReceive.systemFixed.Start )
      { S7_Templates := "[str_type := String, return_type := Int]" } LEN(IN := #mpSerialNumber, OUT => #tempSerialLength)
      wire#w1
      { S7_Templates := "SrcType := String" } NE_Contact(in1 := #mpSerialNumber, in2 := #statSerialOutput)
      wire#w2
      S_Coil( #stateAlarm.serialnumbermismatch )
   END_RUNG
   RUNG wire#w1
      { S7_Templates := "SrcType := Int" } LT_Contact(in1 := #tempSerialLength, in2 := 1)
   END_RUNG wire#w2
   // the same network as SCL:
   #_w1 := NOT #OpModeUserInterfaceOut.opmodeStatus.dryRunActive AND #aux.runSequence AND #aux.dataStrobed AND #statDataExchangeReceive.systemFixed.Start;
   LEN(EN := #_w1, IN := #mpSerialNumber, OUT => #tempSerialLength, ENO => #_w2);
   IF #_w2 AND ((#mpSerialNumber <> #statSerialOutput) OR (#tempSerialLength < 1)) THEN
       #stateAlarm.serialnumbermismatch := TRUE;
   END_IF;
END_REGION

REGION Network 18: Run Sequence
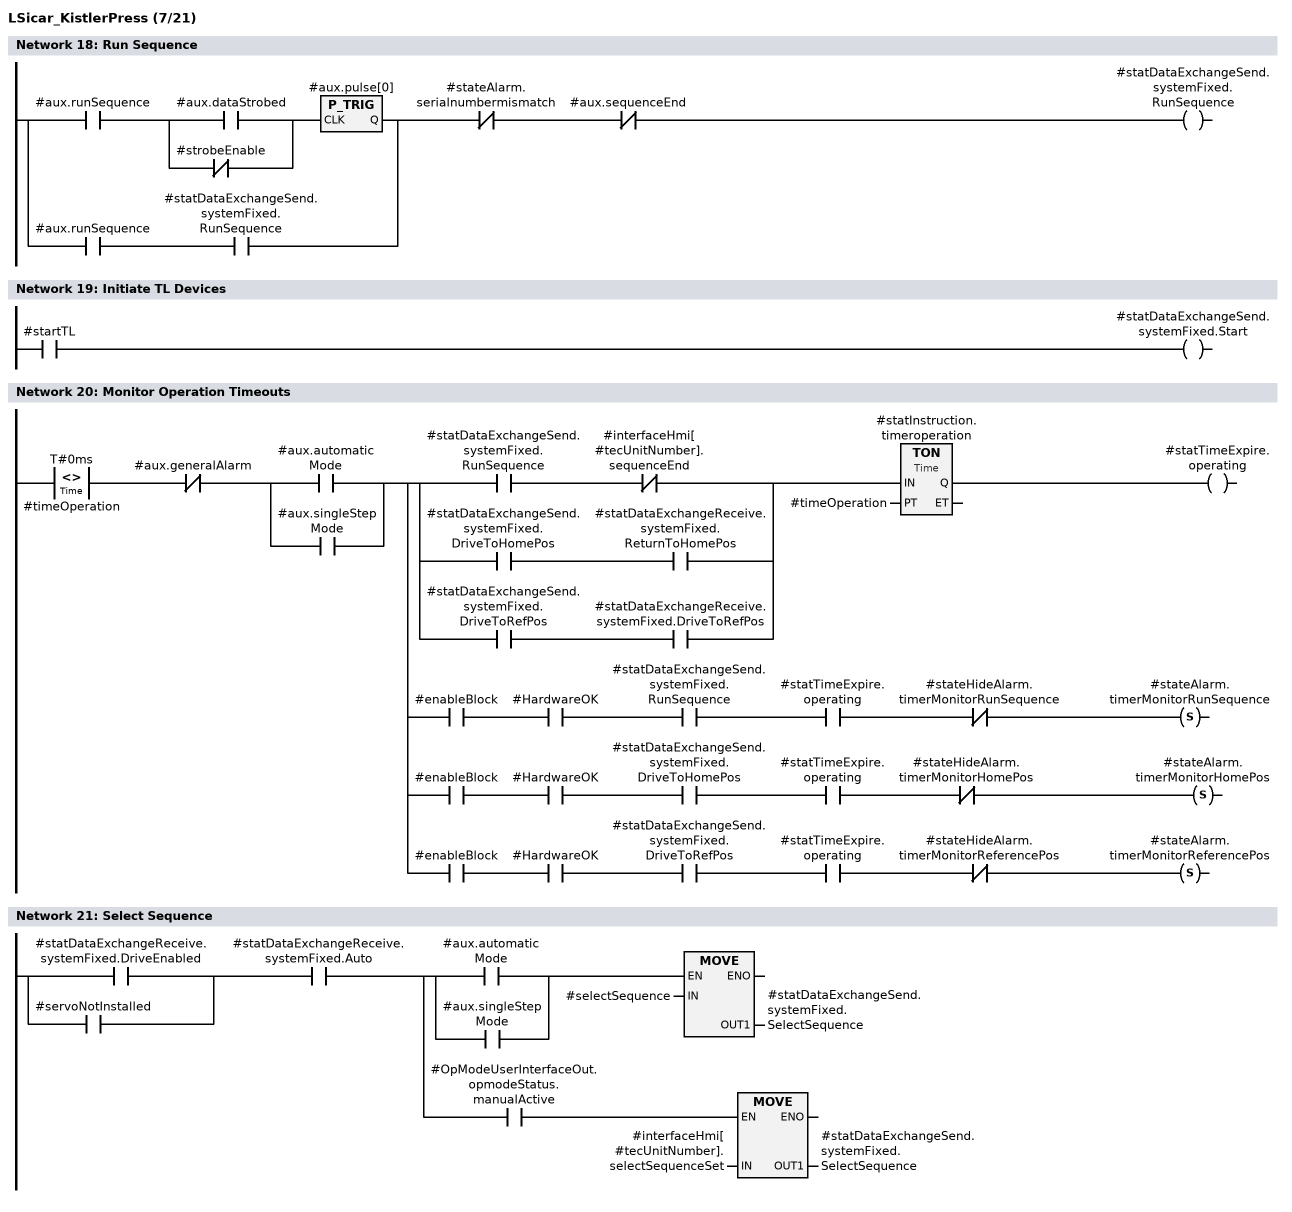
   RUNG wire#powerrail
      Contact( #aux.runSequence )
      wire#w1
      Contact( #aux.dataStrobed )
      wire#w2
      P_Trig( #aux.pulse[0] )
      wire#w3
      I_Contact( #stateAlarm.serialnumbermismatch )
      I_Contact( #aux.sequenceEnd )
      Coil( #statDataExchangeSend.systemFixed.RunSequence )
   END_RUNG
   RUNG wire#w1
      I_Contact( #strobeEnable )
   END_RUNG wire#w2
   RUNG wire#powerrail
      Contact( #aux.runSequence )
      Contact( #statDataExchangeSend.systemFixed.RunSequence )
   END_RUNG wire#w3
   // the same network as SCL:
   #_w1 := #aux.runSequence AND (#aux.dataStrobed OR NOT #strobeEnable);
   #_w2 := #_w1 AND NOT #aux.pulse[0];   // rising edge
   #aux.pulse[0] := #_w1;
   #statDataExchangeSend.systemFixed.RunSequence := (#_w2 OR (#aux.runSequence AND #statDataExchangeSend.systemFixed.RunSequence)) AND NOT #stateAlarm.serialnumbermismatch AND NOT #aux.sequenceEnd;
END_REGION

REGION Network 19: Initiate TL Devices
   RUNG wire#powerrail
      Contact( #startTL )
      Coil( #statDataExchangeSend.systemFixed.Start )
   END_RUNG
   // the same network as SCL:
   #statDataExchangeSend.systemFixed.Start := #startTL;
END_REGION

REGION Network 20: Monitor Operation Timeouts
   RUNG wire#powerrail
      { S7_Templates := "SrcType := Time" } NE_Contact(in1 := T#0ms, in2 := #timeOperation)
      I_Contact( #aux.generalAlarm )
      wire#w1
      Contact( #aux.automaticMode )
      wire#w2
      Contact( #statDataExchangeSend.systemFixed.RunSequence )
      I_Contact( #interfaceHmi[#tecUnitNumber].sequenceEnd )
      wire#w3
      { S7_Templates := "time_type := Time" } #statInstruction.timeroperation.TON(pt := #timeOperation, et =>)
      Coil( #statTimeExpire.operating )
   END_RUNG
   RUNG wire#w1
      Contact( #aux.singleStepMode )
   END_RUNG wire#w2
   RUNG wire#w2
      Contact( #statDataExchangeSend.systemFixed.DriveToHomePos )
      Contact( #statDataExchangeReceive.systemFixed.ReturnToHomePos )
   END_RUNG wire#w3
   RUNG wire#w2
      Contact( #statDataExchangeSend.systemFixed.DriveToRefPos )
      Contact( #statDataExchangeReceive.systemFixed.DriveToRefPos )
   END_RUNG wire#w3
   RUNG wire#w2
      Contact( #enableBlock )
      Contact( #HardwareOK )
      Contact( #statDataExchangeSend.systemFixed.RunSequence )
      Contact( #statTimeExpire.operating )
      I_Contact( #stateHideAlarm.timerMonitorRunSequence )
      S_Coil( #stateAlarm.timerMonitorRunSequence )
   END_RUNG
   RUNG wire#w2
      Contact( #enableBlock )
      Contact( #HardwareOK )
      Contact( #statDataExchangeSend.systemFixed.DriveToHomePos )
      Contact( #statTimeExpire.operating )
      I_Contact( #stateHideAlarm.timerMonitorHomePos )
      S_Coil( #stateAlarm.timerMonitorHomePos )
   END_RUNG
   RUNG wire#w2
      Contact( #enableBlock )
      Contact( #HardwareOK )
      Contact( #statDataExchangeSend.systemFixed.DriveToRefPos )
      Contact( #statTimeExpire.operating )
      I_Contact( #stateHideAlarm.timerMonitorReferencePos )
      S_Coil( #stateAlarm.timerMonitorReferencePos )
   END_RUNG
   // the same network as SCL:
   #_w1 := (T#0ms <> #timeOperation) AND NOT #aux.generalAlarm AND (#aux.automaticMode OR #aux.singleStepMode);
   #statInstruction.timeroperation.TON(IN := #_w1 AND ((#statDataExchangeSend.systemFixed.RunSequence AND NOT #interfaceHmi[#tecUnitNumber].sequenceEnd) OR (#statDataExchangeSend.systemFixed.DriveToHomePos AND #statDataExchangeReceive.systemFixed.ReturnToHomePos) OR (#statDataExchangeSend.systemFixed.DriveToRefPos AND #statDataExchangeReceive.systemFixed.DriveToRefPos)),
                           PT := #timeOperation);
   #statTimeExpire.operating := #statInstruction.timeroperation.Q;
   IF #_w1 AND #enableBlock AND #HardwareOK AND #statDataExchangeSend.systemFixed.RunSequence AND #statTimeExpire.operating AND NOT #stateHideAlarm.timerMonitorRunSequence THEN
       #stateAlarm.timerMonitorRunSequence := TRUE;
   END_IF;
   IF #_w1 AND #enableBlock AND #HardwareOK AND #statDataExchangeSend.systemFixed.DriveToHomePos AND #statTimeExpire.operating AND NOT #stateHideAlarm.timerMonitorHomePos THEN
       #stateAlarm.timerMonitorHomePos := TRUE;
   END_IF;
   IF #_w1 AND #enableBlock AND #HardwareOK AND #statDataExchangeSend.systemFixed.DriveToRefPos AND #statTimeExpire.operating AND NOT #stateHideAlarm.timerMonitorReferencePos THEN
       #stateAlarm.timerMonitorReferencePos := TRUE;
   END_IF;
END_REGION

REGION Network 21: Select Sequence
   RUNG wire#powerrail
      Contact( #statDataExchangeReceive.systemFixed.DriveEnabled )
      wire#w1
      Contact( #statDataExchangeReceive.systemFixed.Auto )
      wire#w2
      Contact( #aux.automaticMode )
      wire#w3
      Move(in := #selectSequence, out1 => #statDataExchangeSend.systemFixed.SelectSequence)
   END_RUNG
   RUNG wire#powerrail
      Contact( #servoNotInstalled )
   END_RUNG wire#w1
   RUNG wire#w2
      Contact( #aux.singleStepMode )
   END_RUNG wire#w3
   RUNG wire#w2
      Contact( #OpModeUserInterfaceOut.opmodeStatus.manualActive )
      Move(in := #interfaceHmi[#tecUnitNumber].selectSequenceSet, out1 => #statDataExchangeSend.systemFixed.SelectSequence)
   END_RUNG
   // the same network as SCL:
   #_w1 := (#statDataExchangeReceive.systemFixed.DriveEnabled OR #servoNotInstalled) AND #statDataExchangeReceive.systemFixed.Auto;
   IF #_w1 AND (#aux.automaticMode OR #aux.singleStepMode) THEN
       #statDataExchangeSend.systemFixed.SelectSequence := #selectSequence;
   END_IF;
   IF #_w1 AND #OpModeUserInterfaceOut.opmodeStatus.manualActive THEN
       #statDataExchangeSend.systemFixed.SelectSequence := #interfaceHmi[#tecUnitNumber].selectSequenceSet;
   END_IF;
END_REGION

REGION Network 22: SeqExtStopReq
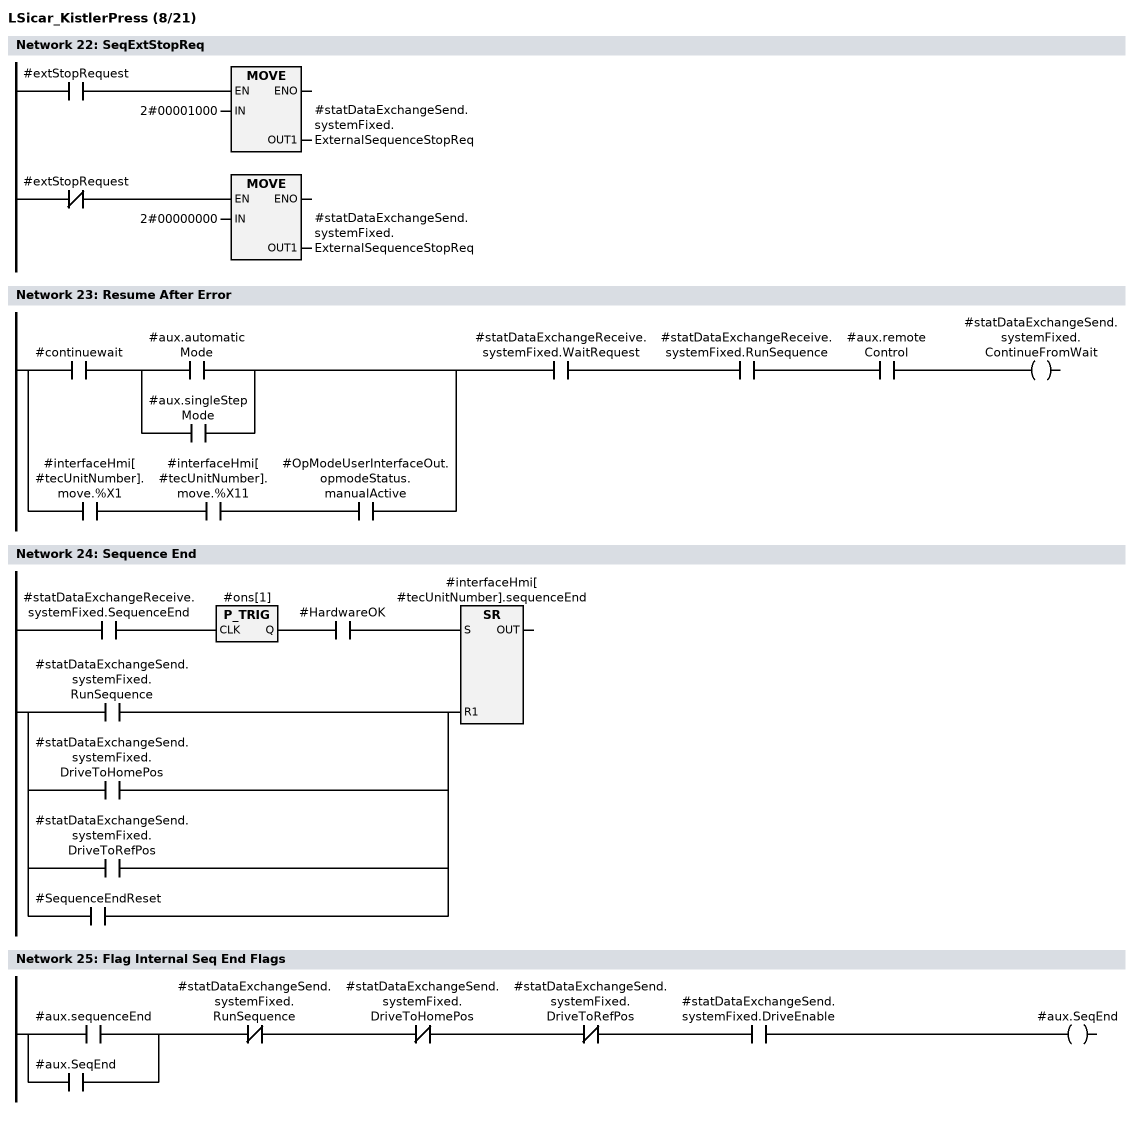
   RUNG wire#powerrail
      Contact( #extStopRequest )
      Move(in := 2#00001000, out1 => #statDataExchangeSend.systemFixed.ExternalSequenceStopReq)
   END_RUNG
   RUNG wire#powerrail
      I_Contact( #extStopRequest )
      Move(in := 2#00000000, out1 => #statDataExchangeSend.systemFixed.ExternalSequenceStopReq)
   END_RUNG
   // the same network as SCL:
   IF #extStopRequest THEN #statDataExchangeSend.systemFixed.ExternalSequenceStopReq := 2#00001000; END_IF;
   IF NOT #extStopRequest THEN
       #statDataExchangeSend.systemFixed.ExternalSequenceStopReq := 2#00000000;
   END_IF;
END_REGION

REGION Network 23: Resume After Error
   RUNG wire#powerrail
      Contact( #continuewait )
      wire#w1
      Contact( #aux.automaticMode )
      wire#w2
      Contact( #statDataExchangeReceive.systemFixed.WaitRequest )
      Contact( #statDataExchangeReceive.systemFixed.RunSequence )
      Contact( #aux.remoteControl )
      Coil( #statDataExchangeSend.systemFixed.ContinueFromWait )
   END_RUNG
   RUNG wire#w1
      Contact( #aux.singleStepMode )
   END_RUNG wire#w2
   RUNG wire#powerrail
      Contact( #interfaceHmi[#tecUnitNumber].move.%X1 )
      Contact( #interfaceHmi[#tecUnitNumber].move.%X11 )
      Contact( #OpModeUserInterfaceOut.opmodeStatus.manualActive )
   END_RUNG wire#w2
   // the same network as SCL:
   #statDataExchangeSend.systemFixed.ContinueFromWait := ((#continuewait AND (#aux.automaticMode OR #aux.singleStepMode)) OR (#interfaceHmi[#tecUnitNumber].move.%X1 AND #interfaceHmi[#tecUnitNumber].move.%X11 AND #OpModeUserInterfaceOut.opmodeStatus.manualActive)) AND #statDataExchangeReceive.systemFixed.WaitRequest AND #statDataExchangeReceive.systemFixed.RunSequence AND #aux.remoteControl;
END_REGION

REGION Network 24: Sequence End
   RUNG wire#powerrail
      Contact( #statDataExchangeReceive.systemFixed.SequenceEnd )
      P_Trig( #ons[1] )
      Contact( #HardwareOK )
      S_SR(operand := #interfaceHmi[#tecUnitNumber].sequenceEnd, r1 := wire#w1)
   END_RUNG
   RUNG wire#powerrail
      Contact( #statDataExchangeSend.systemFixed.RunSequence )
   END_RUNG wire#w1
   RUNG wire#powerrail
      Contact( #statDataExchangeSend.systemFixed.DriveToHomePos )
   END_RUNG wire#w1
   RUNG wire#powerrail
      Contact( #statDataExchangeSend.systemFixed.DriveToRefPos )
   END_RUNG wire#w1
   RUNG wire#powerrail
      Contact( #SequenceEndReset )
   END_RUNG wire#w1
   // the same network as SCL:
   #_w1 := #statDataExchangeReceive.systemFixed.SequenceEnd AND NOT #ons[1];   // rising edge
   #ons[1] := #statDataExchangeReceive.systemFixed.SequenceEnd;
   IF #_w1 AND #HardwareOK THEN
       #interfaceHmi[#tecUnitNumber].sequenceEnd := TRUE;   // SR flip-flop
   END_IF;
   IF #statDataExchangeSend.systemFixed.RunSequence OR #statDataExchangeSend.systemFixed.DriveToHomePos OR #statDataExchangeSend.systemFixed.DriveToRefPos OR #SequenceEndReset THEN
       #interfaceHmi[#tecUnitNumber].sequenceEnd := FALSE;
   END_IF;
END_REGION

REGION Network 25: Flag Internal Seq End Flags
   RUNG wire#powerrail
      Contact( #aux.sequenceEnd )
      wire#w1
      I_Contact( #statDataExchangeSend.systemFixed.RunSequence )
      I_Contact( #statDataExchangeSend.systemFixed.DriveToHomePos )
      I_Contact( #statDataExchangeSend.systemFixed.DriveToRefPos )
      Contact( #statDataExchangeSend.systemFixed.DriveEnable )
      Coil( #aux.SeqEnd )
   END_RUNG
   RUNG wire#powerrail
      Contact( #aux.SeqEnd )
   END_RUNG wire#w1
   // the same network as SCL:
   #aux.SeqEnd := (#aux.sequenceEnd OR #aux.SeqEnd) AND NOT #statDataExchangeSend.systemFixed.RunSequence AND NOT #statDataExchangeSend.systemFixed.DriveToHomePos AND NOT #statDataExchangeSend.systemFixed.DriveToRefPos AND #statDataExchangeSend.systemFixed.DriveEnable;
END_REGION

REGION Network 26: ReturnHomePos
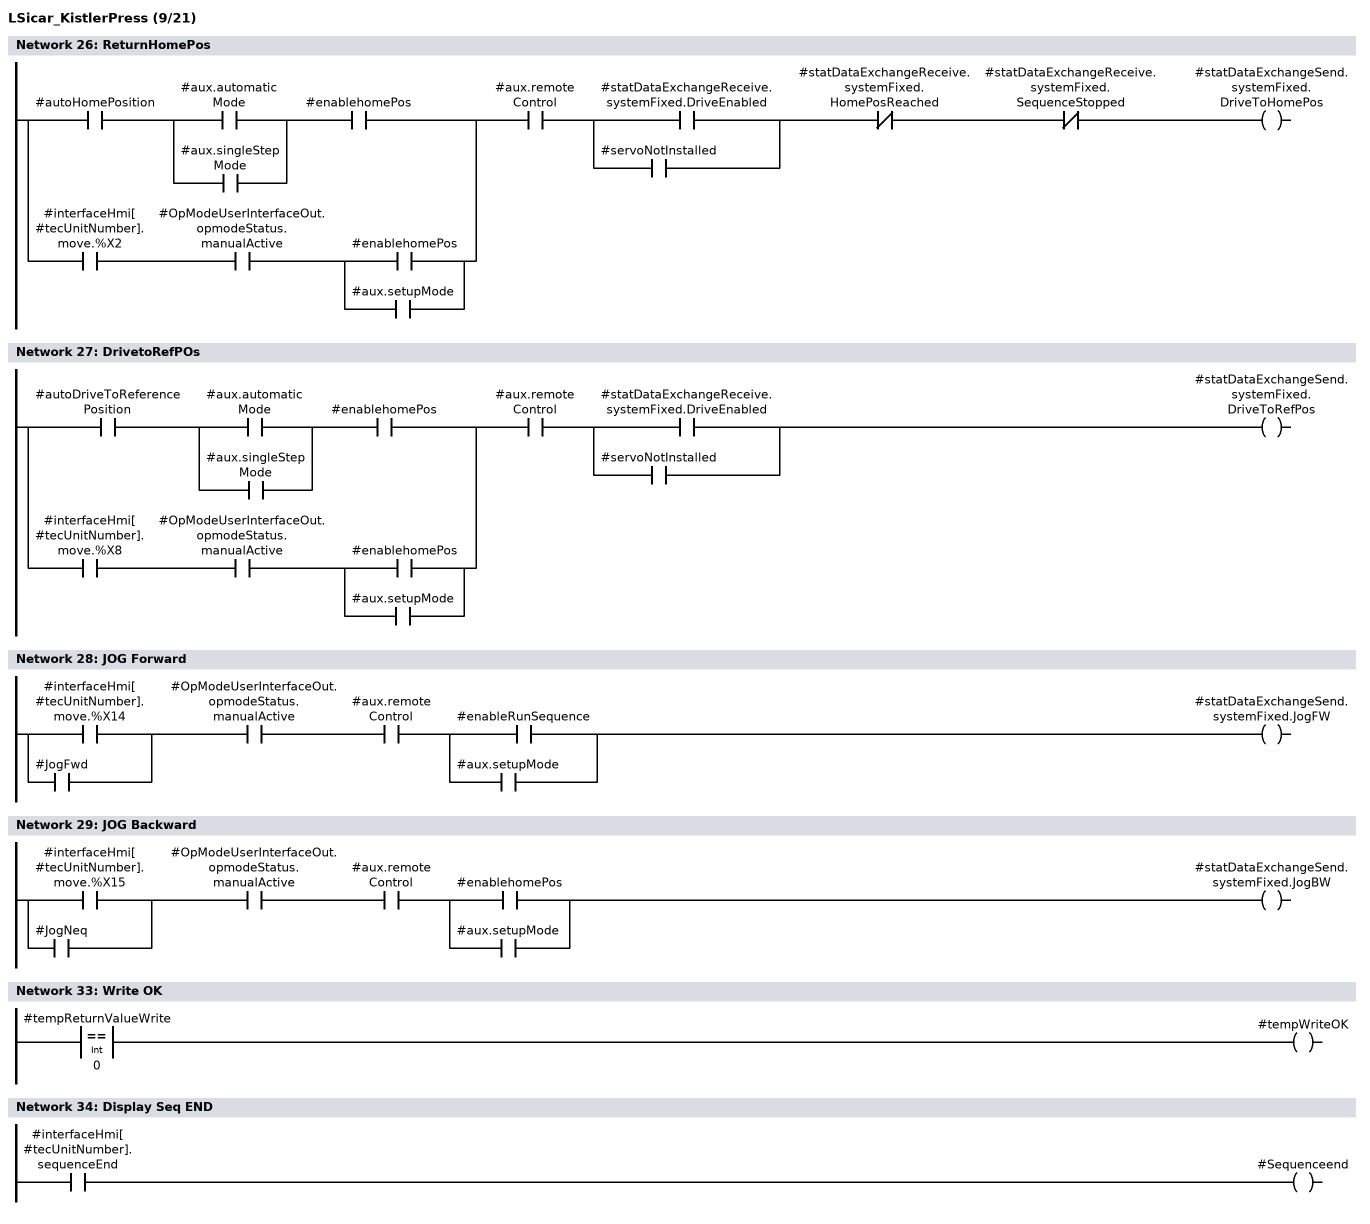
   RUNG wire#powerrail
      Contact( #autoHomePosition )
      wire#w1
      Contact( #aux.automaticMode )
      wire#w2
      Contact( #enablehomePos )
      wire#w3
      Contact( #aux.remoteControl )
      wire#w5
      Contact( #statDataExchangeReceive.systemFixed.DriveEnabled )
      wire#w6
      I_Contact( #statDataExchangeReceive.systemFixed.HomePosReached )
      I_Contact( #statDataExchangeReceive.systemFixed.SequenceStopped )
      Coil( #statDataExchangeSend.systemFixed.DriveToHomePos )
   END_RUNG
   RUNG wire#w1
      Contact( #aux.singleStepMode )
   END_RUNG wire#w2
   RUNG wire#powerrail
      Contact( #interfaceHmi[#tecUnitNumber].move.%X2 )
      Contact( #OpModeUserInterfaceOut.opmodeStatus.manualActive )
      wire#w4
      Contact( #enablehomePos )
   END_RUNG wire#w3
   RUNG wire#w4
      Contact( #aux.setupMode )
   END_RUNG wire#w3
   RUNG wire#w5
      Contact( #servoNotInstalled )
   END_RUNG wire#w6
   // the same network as SCL:
   #statDataExchangeSend.systemFixed.DriveToHomePos := ((#autoHomePosition AND (#aux.automaticMode OR #aux.singleStepMode) AND #enablehomePos) OR (#interfaceHmi[#tecUnitNumber].move.%X2 AND #OpModeUserInterfaceOut.opmodeStatus.manualActive AND (#enablehomePos OR #aux.setupMode))) AND #aux.remoteControl AND (#statDataExchangeReceive.systemFixed.DriveEnabled OR #servoNotInstalled) AND NOT #statDataExchangeReceive.systemFixed.HomePosReached AND NOT #statDataExchangeReceive.systemFixed.SequenceStopped;
END_REGION

REGION Network 27: DrivetoRefPOs
   RUNG wire#powerrail
      Contact( #autoDriveToReferencePosition )
      wire#w1
      Contact( #aux.automaticMode )
      wire#w2
      Contact( #enablehomePos )
      wire#w3
      Contact( #aux.remoteControl )
      wire#w5
      Contact( #statDataExchangeReceive.systemFixed.DriveEnabled )
      wire#w6
      Coil( #statDataExchangeSend.systemFixed.DriveToRefPos )
   END_RUNG
   RUNG wire#w1
      Contact( #aux.singleStepMode )
   END_RUNG wire#w2
   RUNG wire#powerrail
      Contact( #interfaceHmi[#tecUnitNumber].move.%X8 )
      Contact( #OpModeUserInterfaceOut.opmodeStatus.manualActive )
      wire#w4
      Contact( #enablehomePos )
   END_RUNG wire#w3
   RUNG wire#w4
      Contact( #aux.setupMode )
   END_RUNG wire#w3
   RUNG wire#w5
      Contact( #servoNotInstalled )
   END_RUNG wire#w6
   // the same network as SCL:
   #statDataExchangeSend.systemFixed.DriveToRefPos := ((#autoDriveToReferencePosition AND (#aux.automaticMode OR #aux.singleStepMode) AND #enablehomePos) OR (#interfaceHmi[#tecUnitNumber].move.%X8 AND #OpModeUserInterfaceOut.opmodeStatus.manualActive AND (#enablehomePos OR #aux.setupMode))) AND #aux.remoteControl AND (#statDataExchangeReceive.systemFixed.DriveEnabled OR #servoNotInstalled);
END_REGION

REGION Network 28: JOG Forward
   RUNG wire#powerrail
      Contact( #interfaceHmi[#tecUnitNumber].move.%X14 )
      wire#w1
      Contact( #OpModeUserInterfaceOut.opmodeStatus.manualActive )
      Contact( #aux.remoteControl )
      wire#w2
      Contact( #enableRunSequence )
      wire#w3
      Coil( #statDataExchangeSend.systemFixed.JogFW )
   END_RUNG
   RUNG wire#powerrail
      Contact( #JogFwd )
   END_RUNG wire#w1
   RUNG wire#w2
      Contact( #aux.setupMode )
   END_RUNG wire#w3
   // the same network as SCL:
   #statDataExchangeSend.systemFixed.JogFW := (#interfaceHmi[#tecUnitNumber].move.%X14 OR #JogFwd) AND #OpModeUserInterfaceOut.opmodeStatus.manualActive AND #aux.remoteControl AND (#enableRunSequence OR #aux.setupMode);
END_REGION

REGION Network 29: JOG Backward
   RUNG wire#powerrail
      Contact( #interfaceHmi[#tecUnitNumber].move.%X15 )
      wire#w1
      Contact( #OpModeUserInterfaceOut.opmodeStatus.manualActive )
      Contact( #aux.remoteControl )
      wire#w2
      Contact( #enablehomePos )
      wire#w3
      Coil( #statDataExchangeSend.systemFixed.JogBW )
   END_RUNG
   RUNG wire#powerrail
      Contact( #JogNeq )
   END_RUNG wire#w1
   RUNG wire#w2
      Contact( #aux.setupMode )
   END_RUNG wire#w3
   // the same network as SCL:
   #statDataExchangeSend.systemFixed.JogBW := (#interfaceHmi[#tecUnitNumber].move.%X15 OR #JogNeq) AND #OpModeUserInterfaceOut.opmodeStatus.manualActive AND #aux.remoteControl AND (#enablehomePos OR #aux.setupMode);
END_REGION

REGION Network 30 (SCL): Map Incoming Field Bus data for the 200 bytes
   // Jog Speed
   #tempValue := SWAP(REAL_TO_DWORD(#interfaceHmi[#tecUnitNumber].serverJogSpeedSet));
   #statDataExchangeSend.userDefinedOutData[20] := #tempValue.%B0;
   #statDataExchangeSend.userDefinedOutData[21] := #tempValue.%B1;
   #statDataExchangeSend.userDefinedOutData[22] := #tempValue.%B2;
   #statDataExchangeSend.userDefinedOutData[23] := #tempValue.%B3;

   // Jog Max Force
   #tempValue := SWAP(REAL_TO_DWORD(#interfaceHmi[#tecUnitNumber].serverJogMaxForceSet));
   #statDataExchangeSend.userDefinedOutData[24] := #tempValue.%B0;
   #statDataExchangeSend.userDefinedOutData[25] := #tempValue.%B1;
   #statDataExchangeSend.userDefinedOutData[26] := #tempValue.%B2;
   #statDataExchangeSend.userDefinedOutData[27] := #tempValue.%B3;

   // Serial Number
   #tempString := #mpSerialNumber;
   FOR #statSerialByteIndex := 28 TO 51 DO
       #statStringIndex := #statSerialByteIndex - 27;
       #statDataExchangeSend.userDefinedOutData[#statSerialByteIndex] := CHAR_TO_BYTE(#tempString[#statStringIndex]);
   END_FOR;

   // Universal Variables
   #tempDint := 32;
   FOR #i := 0 TO 9 DO
       #tempDword := REAL_TO_DWORD(#parameters.universalvariables[#i]);
       #tempErrorValue := Serialize(SRC_VARIABLE := #tempDword,
                                    DEST_ARRAY => #statDataExchangeSend.userDefinedOutData,
                                    POS := #tempDint);
       #tempDint := #tempDint + 4;
   END_FOR;
END_REGION

REGION Network 31 (SCL): Map Digital Signals
   #statDataExchangeSend.systemFixed.UNI0 := #parameters.UNI_in[0];
   #statDataExchangeSend.systemFixed.UNI1 := #parameters.UNI_in[1];
   #statDataExchangeSend.systemFixed.UNI2 := #parameters.UNI_in[2];
   #statDataExchangeSend.systemFixed.UNI3 := #parameters.UNI_in[3];
   #statDataExchangeSend.systemFixed.UNI4 := #parameters.UNI_in[4];
   #statDataExchangeSend.systemFixed.UNI5 := #parameters.UNI_in[5];
   #statDataExchangeSend.systemFixed.UNI6 := #parameters.UNI_in[6];
   #statDataExchangeSend.systemFixed.UNI7 := #parameters.UNI_in[7];
END_REGION

REGION Network 32 (SCL): Write Raw Data to Kislter
       #tempReturnValueWrite := DPWR_DAT(LADDR := #hardwareID2, RECORD:= #statDataExchangeSend);    // Read from Kistler
END_REGION

REGION Network 33: Write OK
   RUNG wire#powerrail
      { S7_Templates := "SrcType := Int" } EQ_Contact(in1 := #tempReturnValueWrite, in2 := 0)
      Coil( #tempWriteOK )
   END_RUNG
   // the same network as SCL:
   #tempWriteOK := #tempReturnValueWrite = 0;
END_REGION

REGION Network 34: Display Seq END
   RUNG wire#powerrail
      Contact( #interfaceHmi[#tecUnitNumber].sequenceEnd )
      Coil( #Sequenceend )
   END_RUNG
   // the same network as SCL:
   #Sequenceend := #interfaceHmi[#tecUnitNumber].sequenceEnd;
END_REGION

REGION Network 35: Map Fixed Fieldbus outputs to internal flags
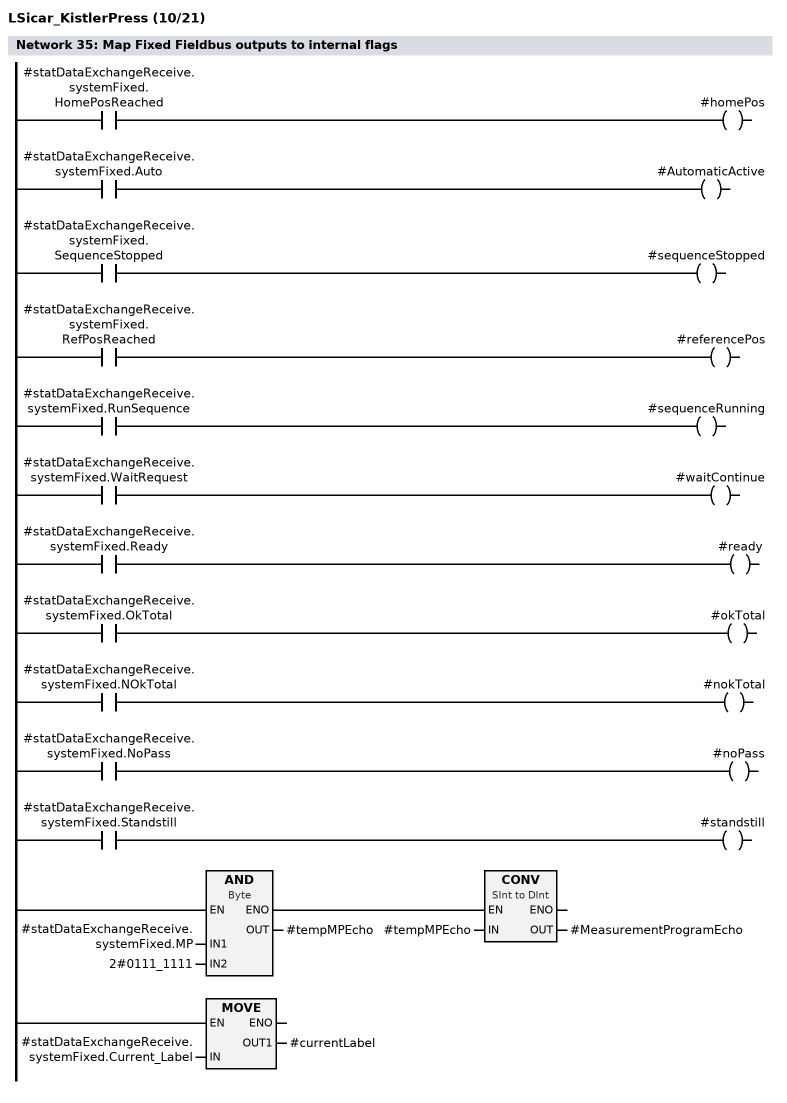
   RUNG wire#powerrail
      Contact( #statDataExchangeReceive.systemFixed.HomePosReached )
      Coil( #homePos )
   END_RUNG
   RUNG wire#powerrail
      Contact( #statDataExchangeReceive.systemFixed.Auto )
      Coil( #AutomaticActive )
   END_RUNG
   RUNG wire#powerrail
      Contact( #statDataExchangeReceive.systemFixed.SequenceStopped )
      Coil( #sequenceStopped )
   END_RUNG
   RUNG wire#powerrail
      Contact( #statDataExchangeReceive.systemFixed.RefPosReached )
      Coil( #referencePos )
   END_RUNG
   RUNG wire#powerrail
      Contact( #statDataExchangeReceive.systemFixed.RunSequence )
      Coil( #sequenceRunning )
   END_RUNG
   RUNG wire#powerrail
      Contact( #statDataExchangeReceive.systemFixed.WaitRequest )
      Coil( #waitContinue )
   END_RUNG
   RUNG wire#powerrail
      Contact( #statDataExchangeReceive.systemFixed.Ready )
      Coil( #ready )
   END_RUNG
   RUNG wire#powerrail
      Contact( #statDataExchangeReceive.systemFixed.OkTotal )
      Coil( #okTotal )
   END_RUNG
   RUNG wire#powerrail
      Contact( #statDataExchangeReceive.systemFixed.NOkTotal )
      Coil( #nokTotal )
   END_RUNG
   RUNG wire#powerrail
      Contact( #statDataExchangeReceive.systemFixed.NoPass )
      Coil( #noPass )
   END_RUNG
   RUNG wire#powerrail
      Contact( #statDataExchangeReceive.systemFixed.Standstill )
      Coil( #standstill )
   END_RUNG
   RUNG wire#powerrail
      { S7_Templates := "SrcType := Byte" } And(in1 := #statDataExchangeReceive.systemFixed.MP, in2 := 2#0111_1111, out => #tempMPEcho)
      { S7_Templates := "[SrcType := SInt, DestType := DInt]" } Convert(in := #tempMPEcho, out => #MeasurementProgramEcho)
   END_RUNG
   RUNG wire#powerrail
      Move(in := #statDataExchangeReceive.systemFixed.Current_Label, out1 => #currentLabel)
   END_RUNG
   // the same network as SCL:
   #homePos := #statDataExchangeReceive.systemFixed.HomePosReached;
   #AutomaticActive := #statDataExchangeReceive.systemFixed.Auto;
   #sequenceStopped := #statDataExchangeReceive.systemFixed.SequenceStopped;
   #referencePos := #statDataExchangeReceive.systemFixed.RefPosReached;
   #sequenceRunning := #statDataExchangeReceive.systemFixed.RunSequence;
   #waitContinue := #statDataExchangeReceive.systemFixed.WaitRequest;
   #ready := #statDataExchangeReceive.systemFixed.Ready;
   #okTotal := #statDataExchangeReceive.systemFixed.OkTotal;
   #nokTotal := #statDataExchangeReceive.systemFixed.NOkTotal;
   #noPass := #statDataExchangeReceive.systemFixed.NoPass;
   #standstill := #statDataExchangeReceive.systemFixed.Standstill;
   #tempMPEcho := #statDataExchangeReceive.systemFixed.MP AND 2#0111_1111;
   #MeasurementProgramEcho := SINT_TO_DINT(#tempMPEcho);
   #currentLabel := #statDataExchangeReceive.systemFixed.Current_Label;
END_REGION

REGION Network 36 (SCL): Process Values Mapping
   // Current Value X
   #tempValue.%B0 := #statDataExchangeReceive.userDefinedOutData[20];
   #tempValue.%B1 := #statDataExchangeReceive.userDefinedOutData[21];
   #tempValue.%B2 := #statDataExchangeReceive.userDefinedOutData[22];
   #tempValue.%B3 := #statDataExchangeReceive.userDefinedOutData[23];
   #pvCurrentValueX := DWORD_TO_REAL(SWAP(#tempValue));

   // Current Value Y
   #tempValue.%B0 := #statDataExchangeReceive.userDefinedOutData[24];
   #tempValue.%B1 := #statDataExchangeReceive.userDefinedOutData[25];
   #tempValue.%B2 := #statDataExchangeReceive.userDefinedOutData[26];
   #tempValue.%B3 := #statDataExchangeReceive.userDefinedOutData[27];
   #pvCurrentValueY := DWORD_TO_REAL(SWAP(#tempValue));

   // Serial Number
   FOR #statSerialByteIndex := 40 TO 63 DO
       #statStringIndex := #statSerialByteIndex - 39;
       #tempString[#statStringIndex] := BYTE_TO_CHAR(#statDataExchangeReceive.userDefinedOutData[#statSerialByteIndex]);
   END_FOR;
   #statSerialOutput := #tempString;

   // Curve XminX
   #tempValue.%B0 := #statDataExchangeReceive.userDefinedOutData[64];
   #tempValue.%B1 := #statDataExchangeReceive.userDefinedOutData[65];
   #tempValue.%B2 := #statDataExchangeReceive.userDefinedOutData[66];
   #tempValue.%B3 := #statDataExchangeReceive.userDefinedOutData[67];
   #pvCurveXminX := DWORD_TO_REAL(SWAP(#tempValue));

   // Curve XmaxX
   #tempValue.%B0 := #statDataExchangeReceive.userDefinedOutData[68];
   #tempValue.%B1 := #statDataExchangeReceive.userDefinedOutData[69];
   #tempValue.%B2 := #statDataExchangeReceive.userDefinedOutData[70];
   #tempValue.%B3 := #statDataExchangeReceive.userDefinedOutData[71];
   #pvCurveXmaxX := DWORD_TO_REAL(SWAP(#tempValue));

   // Curve YminY
   #tempValue.%B0 := #statDataExchangeReceive.userDefinedOutData[72];
   #tempValue.%B1 := #statDataExchangeReceive.userDefinedOutData[73];
   #tempValue.%B2 := #statDataExchangeReceive.userDefinedOutData[74];
   #tempValue.%B3 := #statDataExchangeReceive.userDefinedOutData[75];
   #pvCurveYminY := DWORD_TO_REAL(SWAP(#tempValue));

   // Curve YmaxY
   #tempValue.%B0 := #statDataExchangeReceive.userDefinedOutData[76];
   #tempValue.%B1 := #statDataExchangeReceive.userDefinedOutData[77];
   #tempValue.%B2 := #statDataExchangeReceive.userDefinedOutData[78];
   #tempValue.%B3 := #statDataExchangeReceive.userDefinedOutData[79];
   #pvCurveYmaxY := DWORD_TO_REAL(SWAP(#tempValue));

   // E01 Force
   #tempValue.%B0 := #statDataExchangeReceive.userDefinedOutData[96];
   #tempValue.%B1 := #statDataExchangeReceive.userDefinedOutData[97];
   #tempValue.%B2 := #statDataExchangeReceive.userDefinedOutData[98];
   #tempValue.%B3 := #statDataExchangeReceive.userDefinedOutData[99];
   #customeProcessValues.pv1Force := DWORD_TO_REAL(SWAP(#tempValue));

   // E02 Distance
   #tempValue.%B0 := #statDataExchangeReceive.userDefinedOutData[100];
   #tempValue.%B1 := #statDataExchangeReceive.userDefinedOutData[101];
   #tempValue.%B2 := #statDataExchangeReceive.userDefinedOutData[102];
   #tempValue.%B3 := #statDataExchangeReceive.userDefinedOutData[103];
   #customeProcessValues.pv2Distance := DWORD_TO_REAL(SWAP(#tempValue));

   // E03 Gradient
   #tempValue.%B0 := #statDataExchangeReceive.userDefinedOutData[104];
   #tempValue.%B1 := #statDataExchangeReceive.userDefinedOutData[105];
   #tempValue.%B2 := #statDataExchangeReceive.userDefinedOutData[106];
   #tempValue.%B3 := #statDataExchangeReceive.userDefinedOutData[107];
   #customeProcessValues.pv3Gradient := DWORD_TO_REAL(SWAP(#tempValue));

   // E04 Nopass
   #customeProcessValues.pv4Nopass := #statDataExchangeReceive.userDefinedOutData[108];

   // E05 Unibox
   #customeProcessValues.pv5Unibox := #statDataExchangeReceive.userDefinedOutData[109];

   // E06 Envelope
   #customeProcessValues.pv6Envelope := #statDataExchangeReceive.userDefinedOutData[110];

   // E07 Real
   #tempValue.%B0 := #statDataExchangeReceive.userDefinedOutData[111];
   #tempValue.%B1 := #statDataExchangeReceive.userDefinedOutData[112];
   #tempValue.%B2 := #statDataExchangeReceive.userDefinedOutData[113];
   #tempValue.%B3 := #statDataExchangeReceive.userDefinedOutData[114];
   #customeProcessValues.pv7Real := DWORD_TO_REAL(SWAP(#tempValue));

   // E08 Real
   #tempValue.%B0 := #statDataExchangeReceive.userDefinedOutData[115];
   #tempValue.%B1 := #statDataExchangeReceive.userDefinedOutData[116];
   #tempValue.%B2 := #statDataExchangeReceive.userDefinedOutData[117];
   #tempValue.%B3 := #statDataExchangeReceive.userDefinedOutData[118];
   #customeProcessValues.pv8Real := DWORD_TO_REAL(SWAP(#tempValue));

   // E09 Real
   #tempValue.%B0 := #statDataExchangeReceive.userDefinedOutData[119];
   #tempValue.%B1 := #statDataExchangeReceive.userDefinedOutData[120];
   #tempValue.%B2 := #statDataExchangeReceive.userDefinedOutData[121];
   #tempValue.%B3 := #statDataExchangeReceive.userDefinedOutData[122];
   #customeProcessValues.pv9Real := DWORD_TO_REAL(SWAP(#tempValue));

   // E010 Real
   #tempValue.%B0 := #statDataExchangeReceive.userDefinedOutData[123];
   #tempValue.%B1 := #statDataExchangeReceive.userDefinedOutData[124];
   #tempValue.%B2 := #statDataExchangeReceive.userDefinedOutData[125];
   #tempValue.%B3 := #statDataExchangeReceive.userDefinedOutData[126];
   #customeProcessValues.pv10Real := DWORD_TO_REAL(SWAP(#tempValue));

   // E07 Byte
   #customeProcessValues.pv7Byte := #statDataExchangeReceive.userDefinedOutData[142];

   // E08 Byte
   #customeProcessValues.pv8Byte := #statDataExchangeReceive.userDefinedOutData[143];

   // E09 Byte
   #customeProcessValues.pv9Byte := #statDataExchangeReceive.userDefinedOutData[144];

   // E010 Byte
   #customeProcessValues.pv10Byte := #statDataExchangeReceive.userDefinedOutData[145];
END_REGION

REGION Network 37: Alarms
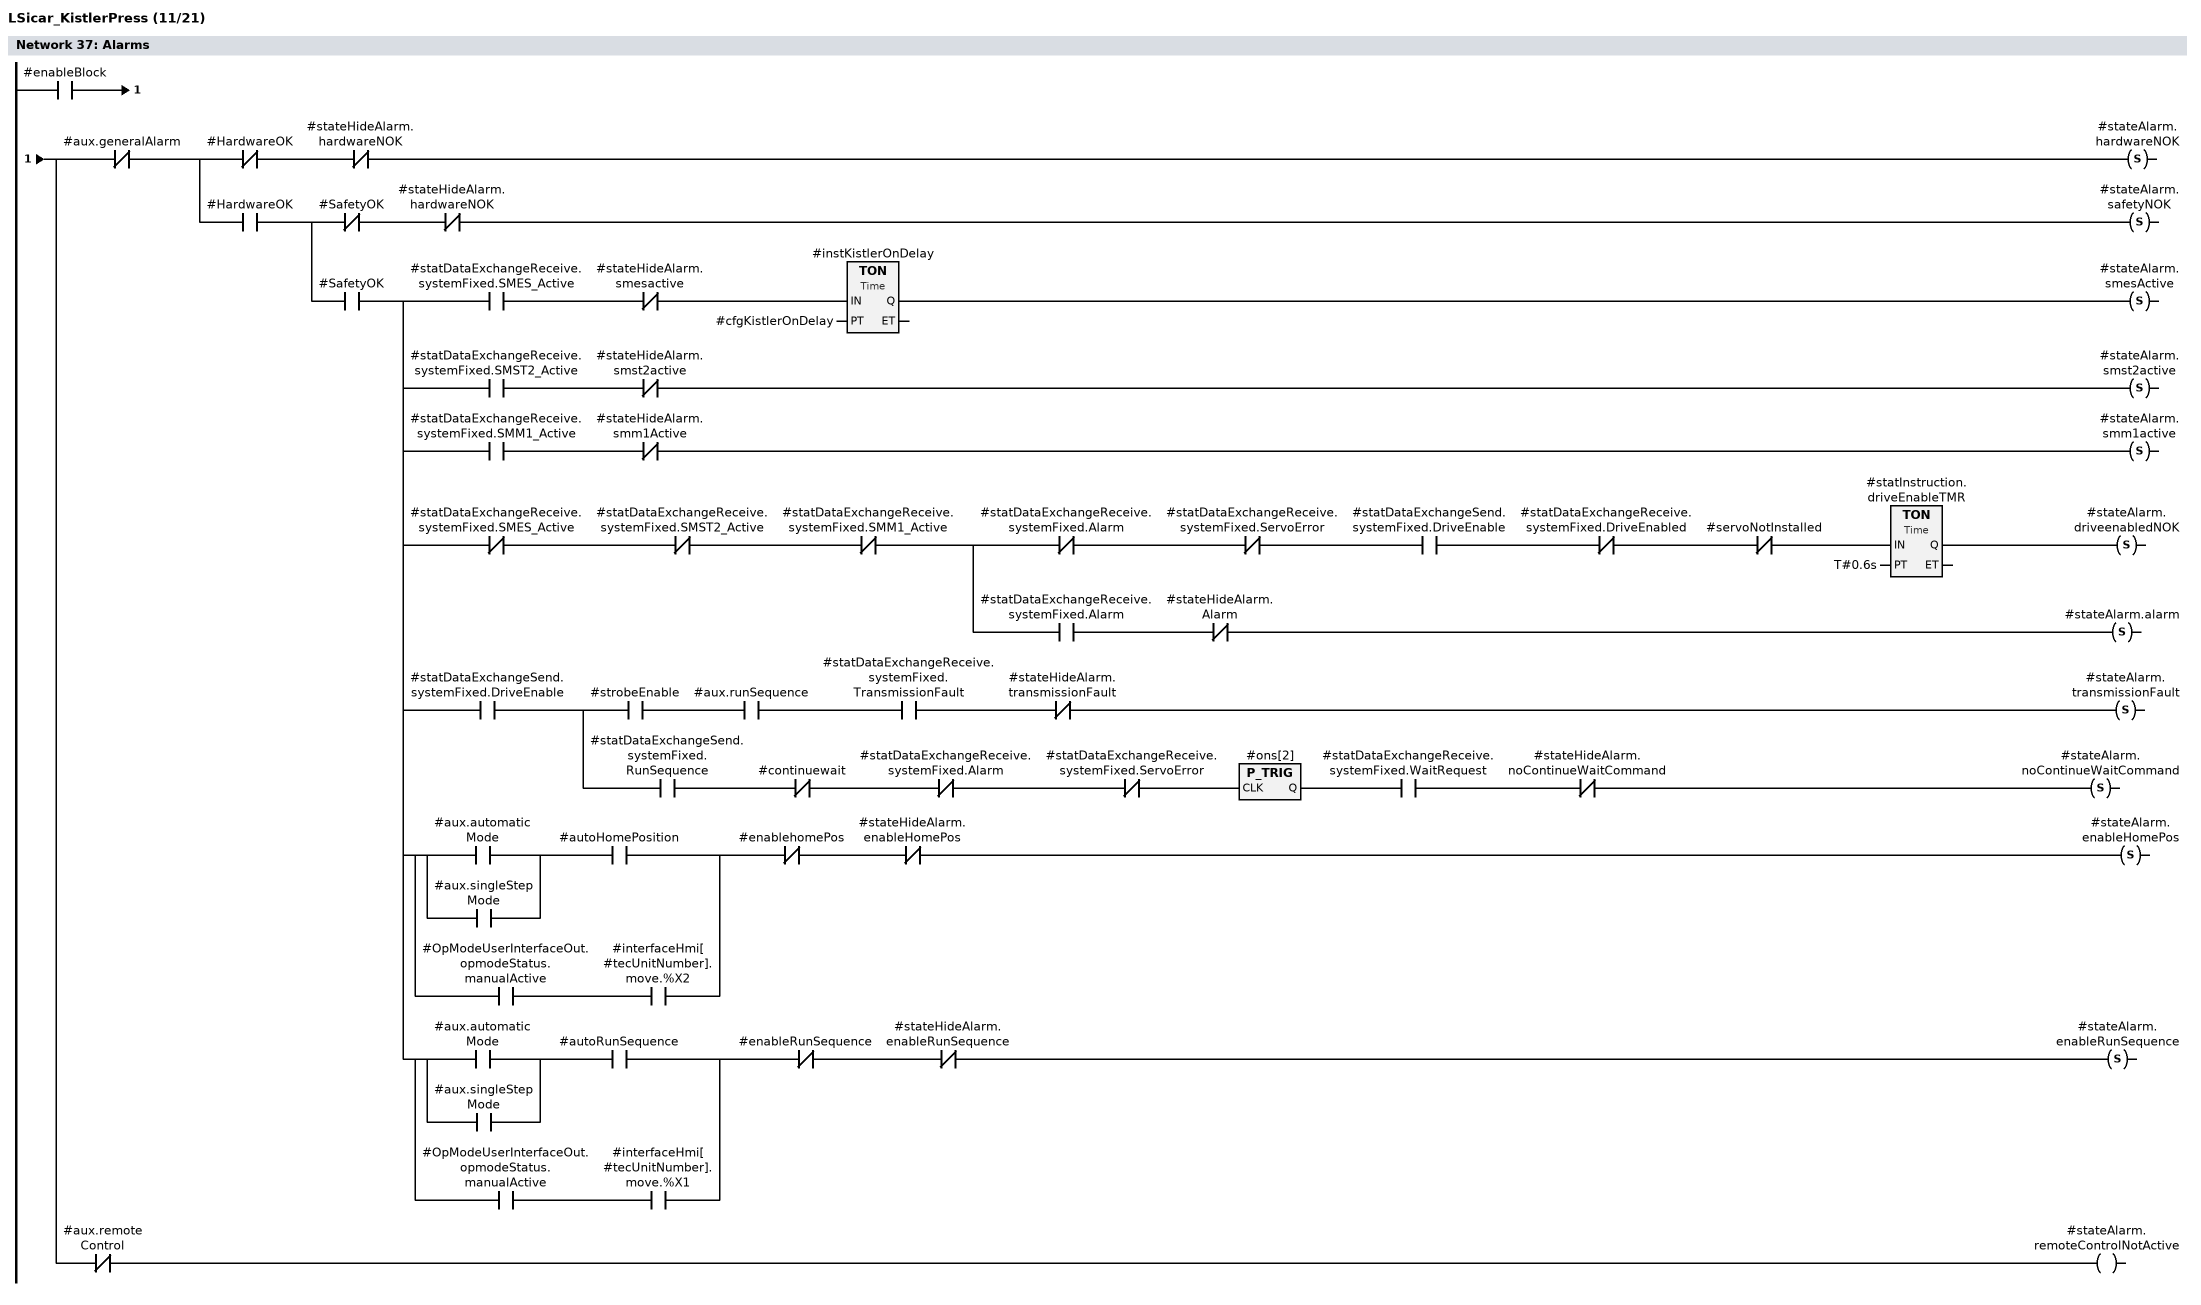
   RUNG wire#powerrail
      Contact( #enableBlock )
      wire#w1
      I_Contact( #aux.generalAlarm )
      wire#w2
      I_Contact( #HardwareOK )
      I_Contact( #stateHideAlarm.hardwareNOK )
      S_Coil( #stateAlarm.hardwareNOK )
   END_RUNG
   RUNG wire#w2
      Contact( #HardwareOK )
      wire#w3
      I_Contact( #SafetyOK )
      I_Contact( #stateHideAlarm.hardwareNOK )
      S_Coil( #stateAlarm.safetyNOK )
   END_RUNG
   RUNG wire#w3
      Contact( #SafetyOK )
      wire#w4
      Contact( #statDataExchangeReceive.systemFixed.SMES_Active )
      I_Contact( #stateHideAlarm.smesactive )
      { S7_Templates := "time_type := Time" } #instKistlerOnDelay.TON(pt := #cfgKistlerOnDelay, et =>)
      S_Coil( #stateAlarm.smesActive )
   END_RUNG
   RUNG wire#w4
      Contact( #statDataExchangeReceive.systemFixed.SMST2_Active )
      I_Contact( #stateHideAlarm.smst2active )
      S_Coil( #stateAlarm.smst2active )
   END_RUNG
   RUNG wire#w4
      Contact( #statDataExchangeReceive.systemFixed.SMM1_Active )
      I_Contact( #stateHideAlarm.smm1Active )
      S_Coil( #stateAlarm.smm1active )
   END_RUNG
   RUNG wire#w4
      I_Contact( #statDataExchangeReceive.systemFixed.SMES_Active )
      I_Contact( #statDataExchangeReceive.systemFixed.SMST2_Active )
      I_Contact( #statDataExchangeReceive.systemFixed.SMM1_Active )
      wire#w5
      I_Contact( #statDataExchangeReceive.systemFixed.Alarm )
      I_Contact( #statDataExchangeReceive.systemFixed.ServoError )
      Contact( #statDataExchangeSend.systemFixed.DriveEnable )
      I_Contact( #statDataExchangeReceive.systemFixed.DriveEnabled )
      I_Contact( #servoNotInstalled )
      { S7_Templates := "time_type := Time" } #statInstruction.driveEnableTMR.TON(pt := T#0.6s, et =>)
      S_Coil( #stateAlarm.driveenabledNOK )
   END_RUNG
   RUNG wire#w5
      Contact( #statDataExchangeReceive.systemFixed.Alarm )
      I_Contact( #stateHideAlarm.Alarm )
      S_Coil( #stateAlarm.alarm )
   END_RUNG
   RUNG wire#w4
      Contact( #statDataExchangeSend.systemFixed.DriveEnable )
      wire#w6
      Contact( #strobeEnable )
      Contact( #aux.runSequence )
      Contact( #statDataExchangeReceive.systemFixed.TransmissionFault )
      I_Contact( #stateHideAlarm.transmissionFault )
      S_Coil( #stateAlarm.transmissionFault )
   END_RUNG
   RUNG wire#w6
      Contact( #statDataExchangeSend.systemFixed.RunSequence )
      I_Contact( #continuewait )
      I_Contact( #statDataExchangeReceive.systemFixed.Alarm )
      I_Contact( #statDataExchangeReceive.systemFixed.ServoError )
      P_Trig( #ons[2] )
      Contact( #statDataExchangeReceive.systemFixed.WaitRequest )
      I_Contact( #stateHideAlarm.noContinueWaitCommand )
      S_Coil( #stateAlarm.noContinueWaitCommand )
   END_RUNG
   RUNG wire#w4
      Contact( #aux.automaticMode )
      wire#w7
      Contact( #autoHomePosition )
      wire#w8
      I_Contact( #enablehomePos )
      I_Contact( #stateHideAlarm.enableHomePos )
      S_Coil( #stateAlarm.enableHomePos )
   END_RUNG
   RUNG wire#w4
      Contact( #aux.singleStepMode )
   END_RUNG wire#w7
   RUNG wire#w4
      Contact( #OpModeUserInterfaceOut.opmodeStatus.manualActive )
      Contact( #interfaceHmi[#tecUnitNumber].move.%X2 )
   END_RUNG wire#w8
   RUNG wire#w4
      Contact( #aux.automaticMode )
      wire#w9
      Contact( #autoRunSequence )
      wire#w10
      I_Contact( #enableRunSequence )
      I_Contact( #stateHideAlarm.enableRunSequence )
      S_Coil( #stateAlarm.enableRunSequence )
   END_RUNG
   RUNG wire#w4
      Contact( #aux.singleStepMode )
   END_RUNG wire#w9
   RUNG wire#w4
      Contact( #OpModeUserInterfaceOut.opmodeStatus.manualActive )
      Contact( #interfaceHmi[#tecUnitNumber].move.%X1 )
   END_RUNG wire#w10
   RUNG wire#w1
      I_Contact( #aux.remoteControl )
      Coil( #stateAlarm.remoteControlNotActive )
   END_RUNG
   // the same network as SCL:
   #_w1 := #enableBlock AND NOT #aux.generalAlarm;
   IF #_w1 AND NOT #HardwareOK AND NOT #stateHideAlarm.hardwareNOK THEN
       #stateAlarm.hardwareNOK := TRUE;
   END_IF;
   #_w2 := #_w1 AND #HardwareOK;
   IF #_w2 AND NOT #SafetyOK AND NOT #stateHideAlarm.hardwareNOK THEN #stateAlarm.safetyNOK := TRUE; END_IF;
   #_w3 := #_w2 AND #SafetyOK;
   #instKistlerOnDelay(IN := #_w3 AND #statDataExchangeReceive.systemFixed.SMES_Active AND NOT #stateHideAlarm.smesactive,   // TON
                       PT := #cfgKistlerOnDelay);
   IF #instKistlerOnDelay.Q THEN #stateAlarm.smesActive := TRUE; END_IF;
   IF #_w3 AND #statDataExchangeReceive.systemFixed.SMST2_Active AND NOT #stateHideAlarm.smst2active THEN
       #stateAlarm.smst2active := TRUE;
   END_IF;
   IF #_w3 AND #statDataExchangeReceive.systemFixed.SMM1_Active AND NOT #stateHideAlarm.smm1Active THEN
       #stateAlarm.smm1active := TRUE;
   END_IF;
   #_w4 := #_w3 AND NOT #statDataExchangeReceive.systemFixed.SMES_Active AND NOT #statDataExchangeReceive.systemFixed.SMST2_Active AND NOT #statDataExchangeReceive.systemFixed.SMM1_Active;
   #statInstruction.driveEnableTMR.TON(IN := #_w4 AND NOT #statDataExchangeReceive.systemFixed.Alarm AND NOT #statDataExchangeReceive.systemFixed.ServoError AND #statDataExchangeSend.systemFixed.DriveEnable AND NOT #statDataExchangeReceive.systemFixed.DriveEnabled AND NOT #servoNotInstalled,
                           PT := T#0.6s);
   IF #statInstruction.driveEnableTMR.Q THEN #stateAlarm.driveenabledNOK := TRUE; END_IF;
   IF #_w4 AND #statDataExchangeReceive.systemFixed.Alarm AND NOT #stateHideAlarm.Alarm THEN
       #stateAlarm.alarm := TRUE;
   END_IF;
   #_w5 := #_w3 AND #statDataExchangeSend.systemFixed.DriveEnable;
   IF #_w5 AND #strobeEnable AND #aux.runSequence AND #statDataExchangeReceive.systemFixed.TransmissionFault AND NOT #stateHideAlarm.transmissionFault THEN
       #stateAlarm.transmissionFault := TRUE;
   END_IF;
   #_w6 := #_w5 AND #statDataExchangeSend.systemFixed.RunSequence AND NOT #continuewait AND NOT #statDataExchangeReceive.systemFixed.Alarm AND NOT #statDataExchangeReceive.systemFixed.ServoError;
   #_w7 := #_w6 AND NOT #ons[2];   // rising edge
   #ons[2] := #_w6;
   IF #_w7 AND #statDataExchangeReceive.systemFixed.WaitRequest AND NOT #stateHideAlarm.noContinueWaitCommand THEN
       #stateAlarm.noContinueWaitCommand := TRUE;
   END_IF;
   IF #_w3 AND (((#aux.automaticMode OR #aux.singleStepMode) AND #autoHomePosition) OR (#OpModeUserInterfaceOut.opmodeStatus.manualActive AND #interfaceHmi[#tecUnitNumber].move.%X2)) AND NOT #enablehomePos AND NOT #stateHideAlarm.enableHomePos THEN
       #stateAlarm.enableHomePos := TRUE;
   END_IF;
   IF #_w3 AND (((#aux.automaticMode OR #aux.singleStepMode) AND #autoRunSequence) OR (#OpModeUserInterfaceOut.opmodeStatus.manualActive AND #interfaceHmi[#tecUnitNumber].move.%X1)) AND NOT #enableRunSequence AND NOT #stateHideAlarm.enableRunSequence THEN
       #stateAlarm.enableRunSequence := TRUE;
   END_IF;
   #stateAlarm.remoteControlNotActive := #enableBlock AND NOT #aux.remoteControl;
END_REGION

REGION Network 38 (SCL): Evaluate Internal Alarms
   #statInternalAlarmNoPD := 0;

   FOR #statAlarmByteIndex := 28 TO 35 DO
       #internalFaultCode[(#statAlarmByteIndex - 28) * 8] := #statDataExchangeReceive.userDefinedOutData[#statAlarmByteIndex].%X0;
       #internalFaultCode[(#statAlarmByteIndex - 28) * 8 + 1] := #statDataExchangeReceive.userDefinedOutData[#statAlarmByteIndex].%X1;
       #internalFaultCode[(#statAlarmByteIndex - 28) * 8 + 2] := #statDataExchangeReceive.userDefinedOutData[#statAlarmByteIndex].%X2;
       #internalFaultCode[(#statAlarmByteIndex - 28) * 8 + 3] := #statDataExchangeReceive.userDefinedOutData[#statAlarmByteIndex].%X3;
       #internalFaultCode[(#statAlarmByteIndex - 28) * 8 + 4] := #statDataExchangeReceive.userDefinedOutData[#statAlarmByteIndex].%X4;
       #internalFaultCode[(#statAlarmByteIndex - 28) * 8 + 5] := #statDataExchangeReceive.userDefinedOutData[#statAlarmByteIndex].%X5;
       #internalFaultCode[(#statAlarmByteIndex - 28) * 8 + 6] := #statDataExchangeReceive.userDefinedOutData[#statAlarmByteIndex].%X6;
       #internalFaultCode[(#statAlarmByteIndex - 28) * 8 + 7] := #statDataExchangeReceive.userDefinedOutData[#statAlarmByteIndex].%X7;
   END_FOR;
END_REGION

REGION Network 39: Fault General Alarm
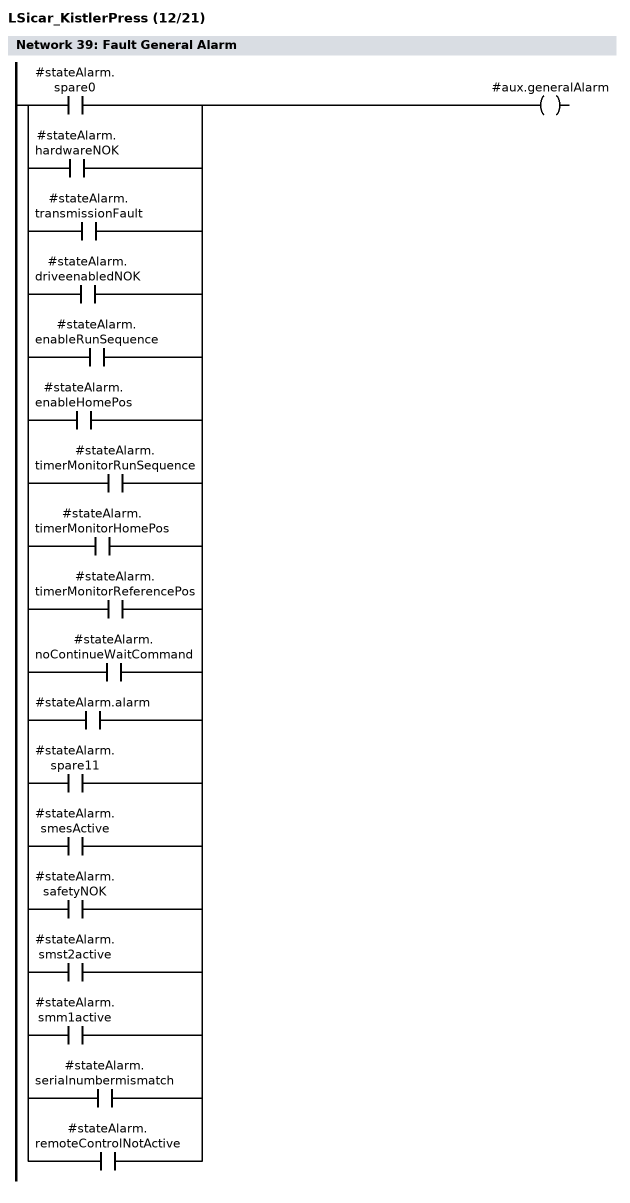
   RUNG wire#powerrail
      Contact( #stateAlarm.spare0 )
      wire#w1
      Coil( #aux.generalAlarm )
   END_RUNG
   RUNG wire#powerrail
      Contact( #stateAlarm.hardwareNOK )
   END_RUNG wire#w1
   RUNG wire#powerrail
      Contact( #stateAlarm.transmissionFault )
   END_RUNG wire#w1
   RUNG wire#powerrail
      Contact( #stateAlarm.driveenabledNOK )
   END_RUNG wire#w1
   RUNG wire#powerrail
      Contact( #stateAlarm.enableRunSequence )
   END_RUNG wire#w1
   RUNG wire#powerrail
      Contact( #stateAlarm.enableHomePos )
   END_RUNG wire#w1
   RUNG wire#powerrail
      Contact( #stateAlarm.timerMonitorRunSequence )
   END_RUNG wire#w1
   RUNG wire#powerrail
      Contact( #stateAlarm.timerMonitorHomePos )
   END_RUNG wire#w1
   RUNG wire#powerrail
      Contact( #stateAlarm.timerMonitorReferencePos )
   END_RUNG wire#w1
   RUNG wire#powerrail
      Contact( #stateAlarm.noContinueWaitCommand )
   END_RUNG wire#w1
   RUNG wire#powerrail
      Contact( #stateAlarm.alarm )
   END_RUNG wire#w1
   RUNG wire#powerrail
      Contact( #stateAlarm.spare11 )
   END_RUNG wire#w1
   RUNG wire#powerrail
      Contact( #stateAlarm.smesActive )
   END_RUNG wire#w1
   RUNG wire#powerrail
      Contact( #stateAlarm.safetyNOK )
   END_RUNG wire#w1
   RUNG wire#powerrail
      Contact( #stateAlarm.smst2active )
   END_RUNG wire#w1
   RUNG wire#powerrail
      Contact( #stateAlarm.smm1active )
   END_RUNG wire#w1
   RUNG wire#powerrail
      Contact( #stateAlarm.serialnumbermismatch )
   END_RUNG wire#w1
   RUNG wire#powerrail
      Contact( #stateAlarm.remoteControlNotActive )
   END_RUNG wire#w1
   // the same network as SCL:
   #aux.generalAlarm := #stateAlarm.spare0 OR #stateAlarm.hardwareNOK OR #stateAlarm.transmissionFault OR #stateAlarm.driveenabledNOK OR #stateAlarm.enableRunSequence OR #stateAlarm.enableHomePos OR #stateAlarm.timerMonitorRunSequence OR #stateAlarm.timerMonitorHomePos OR #stateAlarm.timerMonitorReferencePos OR #stateAlarm.noContinueWaitCommand OR #stateAlarm.alarm OR #stateAlarm.spare11 OR #stateAlarm.smesActive OR #stateAlarm.safetyNOK OR #stateAlarm.smst2active OR #stateAlarm.smm1active OR #stateAlarm.serialnumbermismatch OR #stateAlarm.remoteControlNotActive;
END_REGION

REGION Network 40: Map Alarms to HMI Interface Alarm
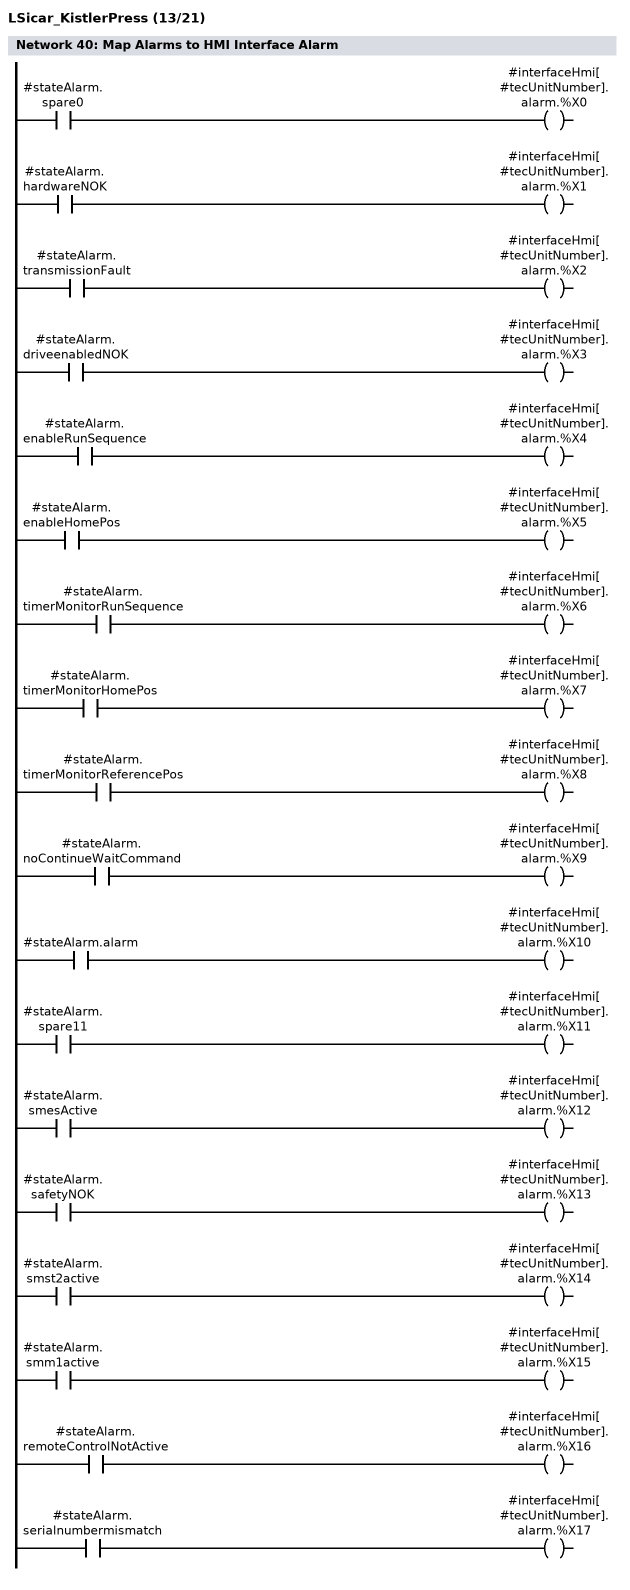
   RUNG wire#powerrail
      Contact( #stateAlarm.spare0 )
      Coil( #interfaceHmi[#tecUnitNumber].alarm.%X0 )
   END_RUNG
   RUNG wire#powerrail
      Contact( #stateAlarm.hardwareNOK )
      Coil( #interfaceHmi[#tecUnitNumber].alarm.%X1 )
   END_RUNG
   RUNG wire#powerrail
      Contact( #stateAlarm.transmissionFault )
      Coil( #interfaceHmi[#tecUnitNumber].alarm.%X2 )
   END_RUNG
   RUNG wire#powerrail
      Contact( #stateAlarm.driveenabledNOK )
      Coil( #interfaceHmi[#tecUnitNumber].alarm.%X3 )
   END_RUNG
   RUNG wire#powerrail
      Contact( #stateAlarm.enableRunSequence )
      Coil( #interfaceHmi[#tecUnitNumber].alarm.%X4 )
   END_RUNG
   RUNG wire#powerrail
      Contact( #stateAlarm.enableHomePos )
      Coil( #interfaceHmi[#tecUnitNumber].alarm.%X5 )
   END_RUNG
   RUNG wire#powerrail
      Contact( #stateAlarm.timerMonitorRunSequence )
      Coil( #interfaceHmi[#tecUnitNumber].alarm.%X6 )
   END_RUNG
   RUNG wire#powerrail
      Contact( #stateAlarm.timerMonitorHomePos )
      Coil( #interfaceHmi[#tecUnitNumber].alarm.%X7 )
   END_RUNG
   RUNG wire#powerrail
      Contact( #stateAlarm.timerMonitorReferencePos )
      Coil( #interfaceHmi[#tecUnitNumber].alarm.%X8 )
   END_RUNG
   RUNG wire#powerrail
      Contact( #stateAlarm.noContinueWaitCommand )
      Coil( #interfaceHmi[#tecUnitNumber].alarm.%X9 )
   END_RUNG
   RUNG wire#powerrail
      Contact( #stateAlarm.alarm )
      Coil( #interfaceHmi[#tecUnitNumber].alarm.%X10 )
   END_RUNG
   RUNG wire#powerrail
      Contact( #stateAlarm.spare11 )
      Coil( #interfaceHmi[#tecUnitNumber].alarm.%X11 )
   END_RUNG
   RUNG wire#powerrail
      Contact( #stateAlarm.smesActive )
      Coil( #interfaceHmi[#tecUnitNumber].alarm.%X12 )
   END_RUNG
   RUNG wire#powerrail
      Contact( #stateAlarm.safetyNOK )
      Coil( #interfaceHmi[#tecUnitNumber].alarm.%X13 )
   END_RUNG
   RUNG wire#powerrail
      Contact( #stateAlarm.smst2active )
      Coil( #interfaceHmi[#tecUnitNumber].alarm.%X14 )
   END_RUNG
   RUNG wire#powerrail
      Contact( #stateAlarm.smm1active )
      Coil( #interfaceHmi[#tecUnitNumber].alarm.%X15 )
   END_RUNG
   RUNG wire#powerrail
      Contact( #stateAlarm.remoteControlNotActive )
      Coil( #interfaceHmi[#tecUnitNumber].alarm.%X16 )
   END_RUNG
   RUNG wire#powerrail
      Contact( #stateAlarm.serialnumbermismatch )
      Coil( #interfaceHmi[#tecUnitNumber].alarm.%X17 )
   END_RUNG
   // the same network as SCL:
   #interfaceHmi[#tecUnitNumber].alarm.%X0 := #stateAlarm.spare0;
   #interfaceHmi[#tecUnitNumber].alarm.%X1 := #stateAlarm.hardwareNOK;
   #interfaceHmi[#tecUnitNumber].alarm.%X2 := #stateAlarm.transmissionFault;
   #interfaceHmi[#tecUnitNumber].alarm.%X3 := #stateAlarm.driveenabledNOK;
   #interfaceHmi[#tecUnitNumber].alarm.%X4 := #stateAlarm.enableRunSequence;
   #interfaceHmi[#tecUnitNumber].alarm.%X5 := #stateAlarm.enableHomePos;
   #interfaceHmi[#tecUnitNumber].alarm.%X6 := #stateAlarm.timerMonitorRunSequence;
   #interfaceHmi[#tecUnitNumber].alarm.%X7 := #stateAlarm.timerMonitorHomePos;
   #interfaceHmi[#tecUnitNumber].alarm.%X8 := #stateAlarm.timerMonitorReferencePos;
   #interfaceHmi[#tecUnitNumber].alarm.%X9 := #stateAlarm.noContinueWaitCommand;
   #interfaceHmi[#tecUnitNumber].alarm.%X10 := #stateAlarm.alarm;
   #interfaceHmi[#tecUnitNumber].alarm.%X11 := #stateAlarm.spare11;
   #interfaceHmi[#tecUnitNumber].alarm.%X12 := #stateAlarm.smesActive;
   #interfaceHmi[#tecUnitNumber].alarm.%X13 := #stateAlarm.safetyNOK;
   #interfaceHmi[#tecUnitNumber].alarm.%X14 := #stateAlarm.smst2active;
   #interfaceHmi[#tecUnitNumber].alarm.%X15 := #stateAlarm.smm1active;
   #interfaceHmi[#tecUnitNumber].alarm.%X16 := #stateAlarm.remoteControlNotActive;
   #interfaceHmi[#tecUnitNumber].alarm.%X17 := #stateAlarm.serialnumbermismatch;
END_REGION

REGION Network 41: Assign PLC Alarm Text List
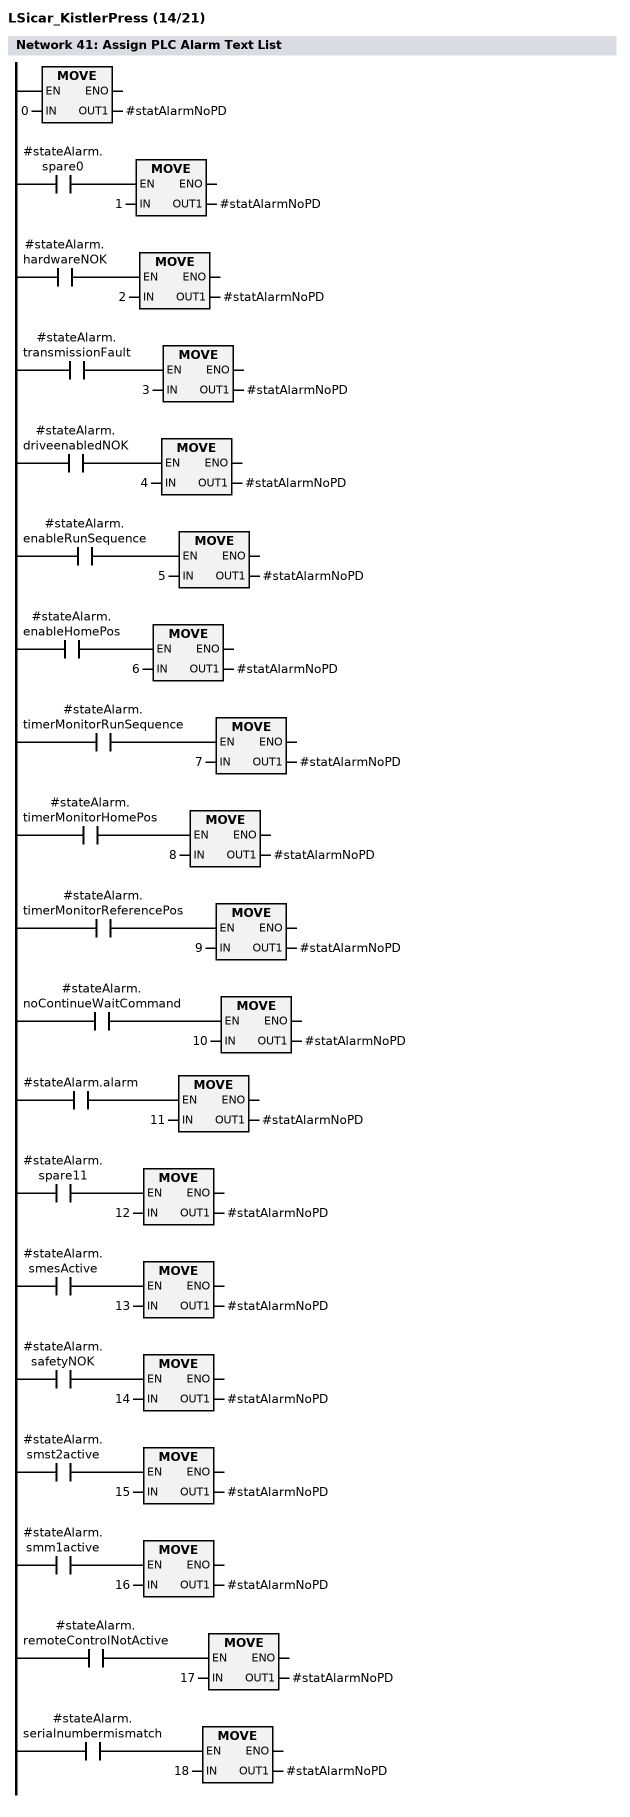
   RUNG wire#powerrail
      Move(in := 0, out1 => #statAlarmNoPD)
   END_RUNG
   RUNG wire#powerrail
      Contact( #stateAlarm.spare0 )
      Move(in := 1, out1 => #statAlarmNoPD)
   END_RUNG
   RUNG wire#powerrail
      Contact( #stateAlarm.hardwareNOK )
      Move(in := 2, out1 => #statAlarmNoPD)
   END_RUNG
   RUNG wire#powerrail
      Contact( #stateAlarm.transmissionFault )
      Move(in := 3, out1 => #statAlarmNoPD)
   END_RUNG
   RUNG wire#powerrail
      Contact( #stateAlarm.driveenabledNOK )
      Move(in := 4, out1 => #statAlarmNoPD)
   END_RUNG
   RUNG wire#powerrail
      Contact( #stateAlarm.enableRunSequence )
      Move(in := 5, out1 => #statAlarmNoPD)
   END_RUNG
   RUNG wire#powerrail
      Contact( #stateAlarm.enableHomePos )
      Move(in := 6, out1 => #statAlarmNoPD)
   END_RUNG
   RUNG wire#powerrail
      Contact( #stateAlarm.timerMonitorRunSequence )
      Move(in := 7, out1 => #statAlarmNoPD)
   END_RUNG
   RUNG wire#powerrail
      Contact( #stateAlarm.timerMonitorHomePos )
      Move(in := 8, out1 => #statAlarmNoPD)
   END_RUNG
   RUNG wire#powerrail
      Contact( #stateAlarm.timerMonitorReferencePos )
      Move(in := 9, out1 => #statAlarmNoPD)
   END_RUNG
   RUNG wire#powerrail
      Contact( #stateAlarm.noContinueWaitCommand )
      Move(in := 10, out1 => #statAlarmNoPD)
   END_RUNG
   RUNG wire#powerrail
      Contact( #stateAlarm.alarm )
      Move(in := 11, out1 => #statAlarmNoPD)
   END_RUNG
   RUNG wire#powerrail
      Contact( #stateAlarm.spare11 )
      Move(in := 12, out1 => #statAlarmNoPD)
   END_RUNG
   RUNG wire#powerrail
      Contact( #stateAlarm.smesActive )
      Move(in := 13, out1 => #statAlarmNoPD)
   END_RUNG
   RUNG wire#powerrail
      Contact( #stateAlarm.safetyNOK )
      Move(in := 14, out1 => #statAlarmNoPD)
   END_RUNG
   RUNG wire#powerrail
      Contact( #stateAlarm.smst2active )
      Move(in := 15, out1 => #statAlarmNoPD)
   END_RUNG
   RUNG wire#powerrail
      Contact( #stateAlarm.smm1active )
      Move(in := 16, out1 => #statAlarmNoPD)
   END_RUNG
   RUNG wire#powerrail
      Contact( #stateAlarm.remoteControlNotActive )
      Move(in := 17, out1 => #statAlarmNoPD)
   END_RUNG
   RUNG wire#powerrail
      Contact( #stateAlarm.serialnumbermismatch )
      Move(in := 18, out1 => #statAlarmNoPD)
   END_RUNG
   // the same network as SCL:
   #statAlarmNoPD := 0;
   IF #stateAlarm.spare0 THEN #statAlarmNoPD := 1; END_IF;
   IF #stateAlarm.hardwareNOK THEN #statAlarmNoPD := 2; END_IF;
   IF #stateAlarm.transmissionFault THEN #statAlarmNoPD := 3; END_IF;
   IF #stateAlarm.driveenabledNOK THEN #statAlarmNoPD := 4; END_IF;
   IF #stateAlarm.enableRunSequence THEN #statAlarmNoPD := 5; END_IF;
   IF #stateAlarm.enableHomePos THEN #statAlarmNoPD := 6; END_IF;
   IF #stateAlarm.timerMonitorRunSequence THEN #statAlarmNoPD := 7; END_IF;
   IF #stateAlarm.timerMonitorHomePos THEN #statAlarmNoPD := 8; END_IF;
   IF #stateAlarm.timerMonitorReferencePos THEN #statAlarmNoPD := 9; END_IF;
   IF #stateAlarm.noContinueWaitCommand THEN #statAlarmNoPD := 10; END_IF;
   IF #stateAlarm.alarm THEN #statAlarmNoPD := 11; END_IF;
   IF #stateAlarm.spare11 THEN #statAlarmNoPD := 12; END_IF;
   IF #stateAlarm.smesActive THEN #statAlarmNoPD := 13; END_IF;
   IF #stateAlarm.safetyNOK THEN #statAlarmNoPD := 14; END_IF;
   IF #stateAlarm.smst2active THEN #statAlarmNoPD := 15; END_IF;
   IF #stateAlarm.smm1active THEN #statAlarmNoPD := 16; END_IF;
   IF #stateAlarm.remoteControlNotActive THEN #statAlarmNoPD := 17; END_IF;
   IF #stateAlarm.serialnumbermismatch THEN #statAlarmNoPD := 18; END_IF;
END_REGION

REGION Network 42: HMI Color Association
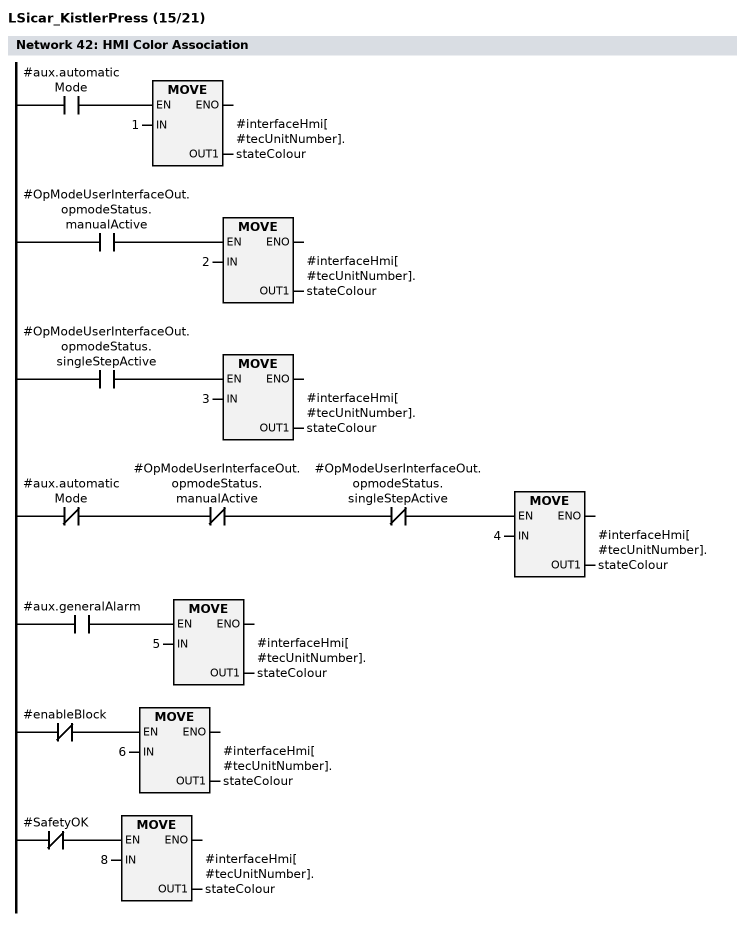
   RUNG wire#powerrail
      Contact( #aux.automaticMode )
      Move(in := 1, out1 => #interfaceHmi[#tecUnitNumber].stateColour)
   END_RUNG
   RUNG wire#powerrail
      Contact( #OpModeUserInterfaceOut.opmodeStatus.manualActive )
      Move(in := 2, out1 => #interfaceHmi[#tecUnitNumber].stateColour)
   END_RUNG
   RUNG wire#powerrail
      Contact( #OpModeUserInterfaceOut.opmodeStatus.singleStepActive )
      Move(in := 3, out1 => #interfaceHmi[#tecUnitNumber].stateColour)
   END_RUNG
   RUNG wire#powerrail
      I_Contact( #aux.automaticMode )
      I_Contact( #OpModeUserInterfaceOut.opmodeStatus.manualActive )
      I_Contact( #OpModeUserInterfaceOut.opmodeStatus.singleStepActive )
      Move(in := 4, out1 => #interfaceHmi[#tecUnitNumber].stateColour)
   END_RUNG
   RUNG wire#powerrail
      Contact( #aux.generalAlarm )
      Move(in := 5, out1 => #interfaceHmi[#tecUnitNumber].stateColour)
   END_RUNG
   RUNG wire#powerrail
      I_Contact( #enableBlock )
      Move(in := 6, out1 => #interfaceHmi[#tecUnitNumber].stateColour)
   END_RUNG
   RUNG wire#powerrail
      I_Contact( #SafetyOK )
      Move(in := 8, out1 => #interfaceHmi[#tecUnitNumber].stateColour)
   END_RUNG
   // the same network as SCL:
   IF #aux.automaticMode THEN #interfaceHmi[#tecUnitNumber].stateColour := 1; END_IF;
   IF #OpModeUserInterfaceOut.opmodeStatus.manualActive THEN
       #interfaceHmi[#tecUnitNumber].stateColour := 2;
   END_IF;
   IF #OpModeUserInterfaceOut.opmodeStatus.singleStepActive THEN
       #interfaceHmi[#tecUnitNumber].stateColour := 3;
   END_IF;
   IF NOT #aux.automaticMode AND NOT #OpModeUserInterfaceOut.opmodeStatus.manualActive AND NOT #OpModeUserInterfaceOut.opmodeStatus.singleStepActive THEN
       #interfaceHmi[#tecUnitNumber].stateColour := 4;
   END_IF;
   IF #aux.generalAlarm THEN #interfaceHmi[#tecUnitNumber].stateColour := 5; END_IF;
   IF NOT #enableBlock THEN #interfaceHmi[#tecUnitNumber].stateColour := 6; END_IF;
   IF NOT #SafetyOK THEN #interfaceHmi[#tecUnitNumber].stateColour := 8; END_IF;
END_REGION

REGION Network 43: HMI state Mapping
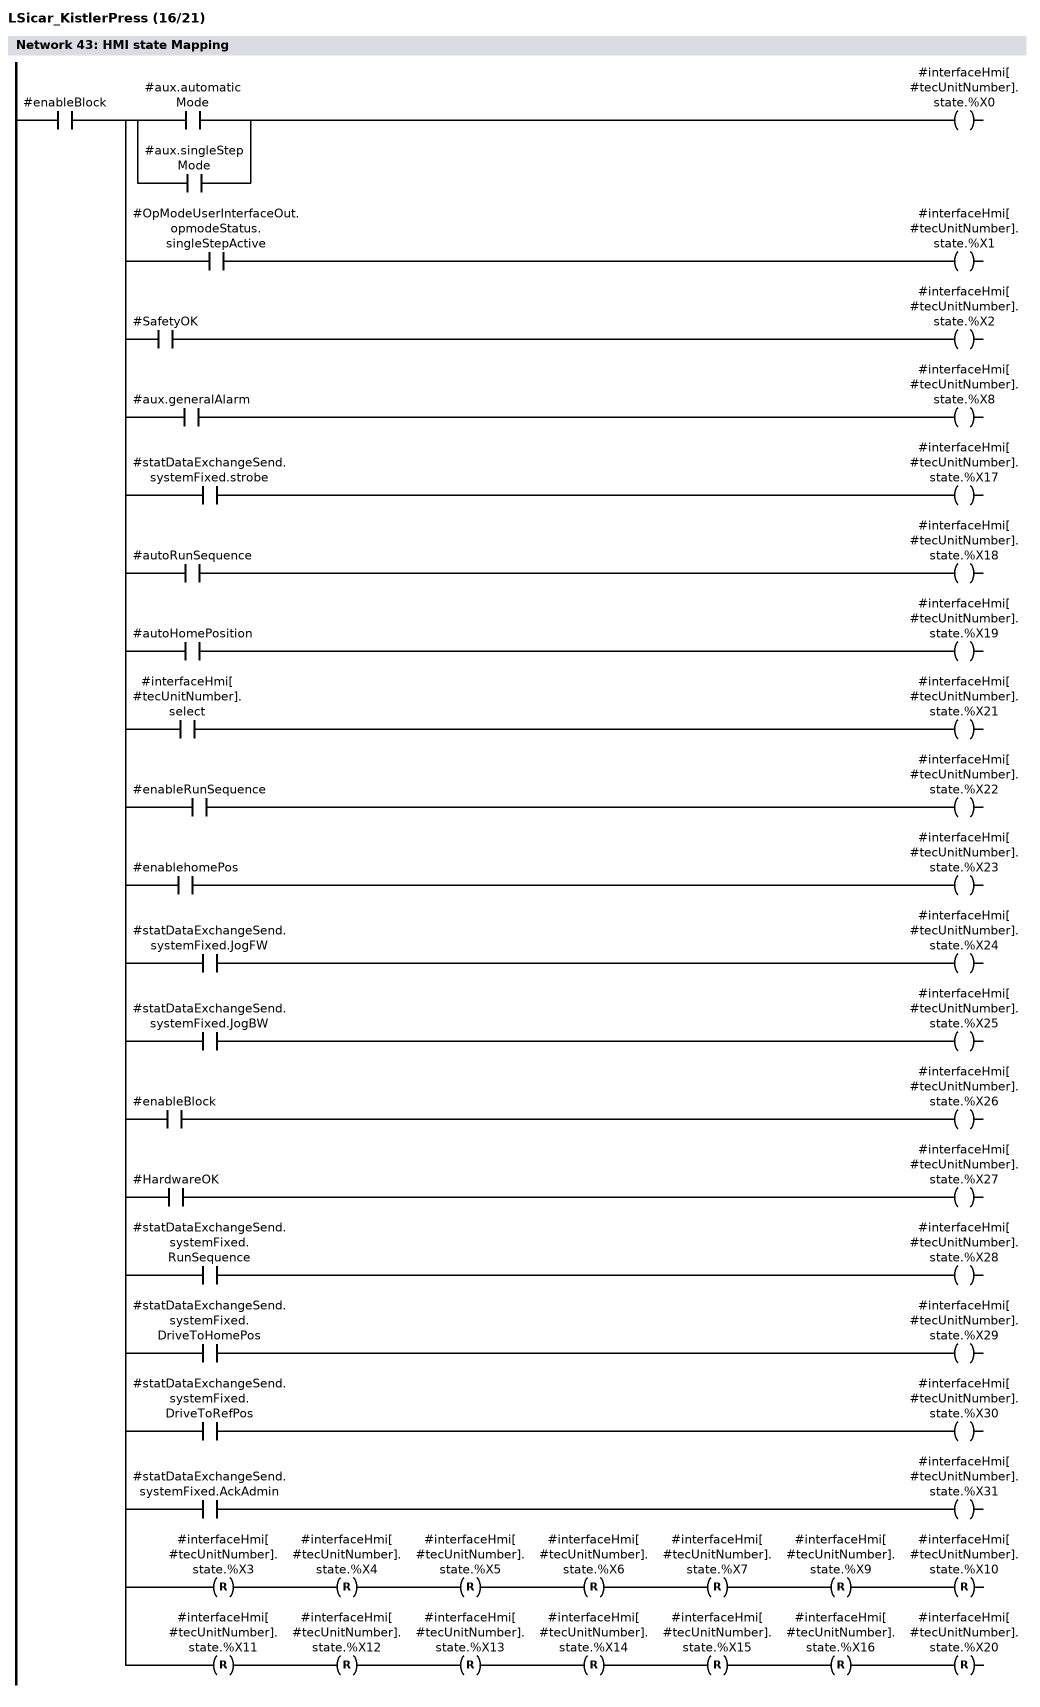
   RUNG wire#powerrail
      Contact( #enableBlock )
      wire#w1
      Contact( #aux.automaticMode )
      wire#w2
      Coil( #interfaceHmi[#tecUnitNumber].state.%X0 )
   END_RUNG
   RUNG wire#w1
      Contact( #aux.singleStepMode )
   END_RUNG wire#w2
   RUNG wire#w1
      Contact( #OpModeUserInterfaceOut.opmodeStatus.singleStepActive )
      Coil( #interfaceHmi[#tecUnitNumber].state.%X1 )
   END_RUNG
   RUNG wire#w1
      Contact( #SafetyOK )
      Coil( #interfaceHmi[#tecUnitNumber].state.%X2 )
   END_RUNG
   RUNG wire#w1
      Contact( #aux.generalAlarm )
      Coil( #interfaceHmi[#tecUnitNumber].state.%X8 )
   END_RUNG
   RUNG wire#w1
      Contact( #statDataExchangeSend.systemFixed.strobe )
      Coil( #interfaceHmi[#tecUnitNumber].state.%X17 )
   END_RUNG
   RUNG wire#w1
      Contact( #autoRunSequence )
      Coil( #interfaceHmi[#tecUnitNumber].state.%X18 )
   END_RUNG
   RUNG wire#w1
      Contact( #autoHomePosition )
      Coil( #interfaceHmi[#tecUnitNumber].state.%X19 )
   END_RUNG
   RUNG wire#w1
      Contact( #interfaceHmi[#tecUnitNumber].select )
      Coil( #interfaceHmi[#tecUnitNumber].state.%X21 )
   END_RUNG
   RUNG wire#w1
      Contact( #enableRunSequence )
      Coil( #interfaceHmi[#tecUnitNumber].state.%X22 )
   END_RUNG
   RUNG wire#w1
      Contact( #enablehomePos )
      Coil( #interfaceHmi[#tecUnitNumber].state.%X23 )
   END_RUNG
   RUNG wire#w1
      Contact( #statDataExchangeSend.systemFixed.JogFW )
      Coil( #interfaceHmi[#tecUnitNumber].state.%X24 )
   END_RUNG
   RUNG wire#w1
      Contact( #statDataExchangeSend.systemFixed.JogBW )
      Coil( #interfaceHmi[#tecUnitNumber].state.%X25 )
   END_RUNG
   RUNG wire#w1
      Contact( #enableBlock )
      Coil( #interfaceHmi[#tecUnitNumber].state.%X26 )
   END_RUNG
   RUNG wire#w1
      Contact( #HardwareOK )
      Coil( #interfaceHmi[#tecUnitNumber].state.%X27 )
   END_RUNG
   RUNG wire#w1
      Contact( #statDataExchangeSend.systemFixed.RunSequence )
      Coil( #interfaceHmi[#tecUnitNumber].state.%X28 )
   END_RUNG
   RUNG wire#w1
      Contact( #statDataExchangeSend.systemFixed.DriveToHomePos )
      Coil( #interfaceHmi[#tecUnitNumber].state.%X29 )
   END_RUNG
   RUNG wire#w1
      Contact( #statDataExchangeSend.systemFixed.DriveToRefPos )
      Coil( #interfaceHmi[#tecUnitNumber].state.%X30 )
   END_RUNG
   RUNG wire#w1
      Contact( #statDataExchangeSend.systemFixed.AckAdmin )
      Coil( #interfaceHmi[#tecUnitNumber].state.%X31 )
   END_RUNG
   RUNG wire#w1
      R_Coil( #interfaceHmi[#tecUnitNumber].state.%X3 )
      R_Coil( #interfaceHmi[#tecUnitNumber].state.%X4 )
      R_Coil( #interfaceHmi[#tecUnitNumber].state.%X5 )
      R_Coil( #interfaceHmi[#tecUnitNumber].state.%X6 )
      R_Coil( #interfaceHmi[#tecUnitNumber].state.%X7 )
      R_Coil( #interfaceHmi[#tecUnitNumber].state.%X9 )
      R_Coil( #interfaceHmi[#tecUnitNumber].state.%X10 )
   END_RUNG
   RUNG wire#w1
      R_Coil( #interfaceHmi[#tecUnitNumber].state.%X11 )
      R_Coil( #interfaceHmi[#tecUnitNumber].state.%X12 )
      R_Coil( #interfaceHmi[#tecUnitNumber].state.%X13 )
      R_Coil( #interfaceHmi[#tecUnitNumber].state.%X14 )
      R_Coil( #interfaceHmi[#tecUnitNumber].state.%X15 )
      R_Coil( #interfaceHmi[#tecUnitNumber].state.%X16 )
      R_Coil( #interfaceHmi[#tecUnitNumber].state.%X20 )
   END_RUNG
   // the same network as SCL:
   #interfaceHmi[#tecUnitNumber].state.%X0 := #enableBlock AND (#aux.automaticMode OR #aux.singleStepMode);
   #interfaceHmi[#tecUnitNumber].state.%X1 := #enableBlock AND #OpModeUserInterfaceOut.opmodeStatus.singleStepActive;
   #interfaceHmi[#tecUnitNumber].state.%X2 := #enableBlock AND #SafetyOK;
   #interfaceHmi[#tecUnitNumber].state.%X8 := #enableBlock AND #aux.generalAlarm;
   #interfaceHmi[#tecUnitNumber].state.%X17 := #enableBlock AND #statDataExchangeSend.systemFixed.strobe;
   #interfaceHmi[#tecUnitNumber].state.%X18 := #enableBlock AND #autoRunSequence;
   #interfaceHmi[#tecUnitNumber].state.%X19 := #enableBlock AND #autoHomePosition;
   #interfaceHmi[#tecUnitNumber].state.%X21 := #enableBlock AND #interfaceHmi[#tecUnitNumber].select;
   #interfaceHmi[#tecUnitNumber].state.%X22 := #enableBlock AND #enableRunSequence;
   #interfaceHmi[#tecUnitNumber].state.%X23 := #enableBlock AND #enablehomePos;
   #interfaceHmi[#tecUnitNumber].state.%X24 := #enableBlock AND #statDataExchangeSend.systemFixed.JogFW;
   #interfaceHmi[#tecUnitNumber].state.%X25 := #enableBlock AND #statDataExchangeSend.systemFixed.JogBW;
   #interfaceHmi[#tecUnitNumber].state.%X26 := #enableBlock AND #enableBlock;
   #interfaceHmi[#tecUnitNumber].state.%X27 := #enableBlock AND #HardwareOK;
   #interfaceHmi[#tecUnitNumber].state.%X28 := #enableBlock AND #statDataExchangeSend.systemFixed.RunSequence;
   #interfaceHmi[#tecUnitNumber].state.%X29 := #enableBlock AND #statDataExchangeSend.systemFixed.DriveToHomePos;
   #interfaceHmi[#tecUnitNumber].state.%X30 := #enableBlock AND #statDataExchangeSend.systemFixed.DriveToRefPos;
   #interfaceHmi[#tecUnitNumber].state.%X31 := #enableBlock AND #statDataExchangeSend.systemFixed.AckAdmin;
   IF #enableBlock THEN
       #interfaceHmi[#tecUnitNumber].state.%X3 := FALSE;
       #interfaceHmi[#tecUnitNumber].state.%X4 := FALSE;
       #interfaceHmi[#tecUnitNumber].state.%X5 := FALSE;
       #interfaceHmi[#tecUnitNumber].state.%X6 := FALSE;
       #interfaceHmi[#tecUnitNumber].state.%X7 := FALSE;
       #interfaceHmi[#tecUnitNumber].state.%X9 := FALSE;
       #interfaceHmi[#tecUnitNumber].state.%X10 := FALSE;
       #interfaceHmi[#tecUnitNumber].state.%X11 := FALSE;
       #interfaceHmi[#tecUnitNumber].state.%X12 := FALSE;
       #interfaceHmi[#tecUnitNumber].state.%X13 := FALSE;
       #interfaceHmi[#tecUnitNumber].state.%X14 := FALSE;
       #interfaceHmi[#tecUnitNumber].state.%X15 := FALSE;
       #interfaceHmi[#tecUnitNumber].state.%X16 := FALSE;
       #interfaceHmi[#tecUnitNumber].state.%X20 := FALSE;
   END_IF;
END_REGION

REGION Network 44: Send Process Values to HMI
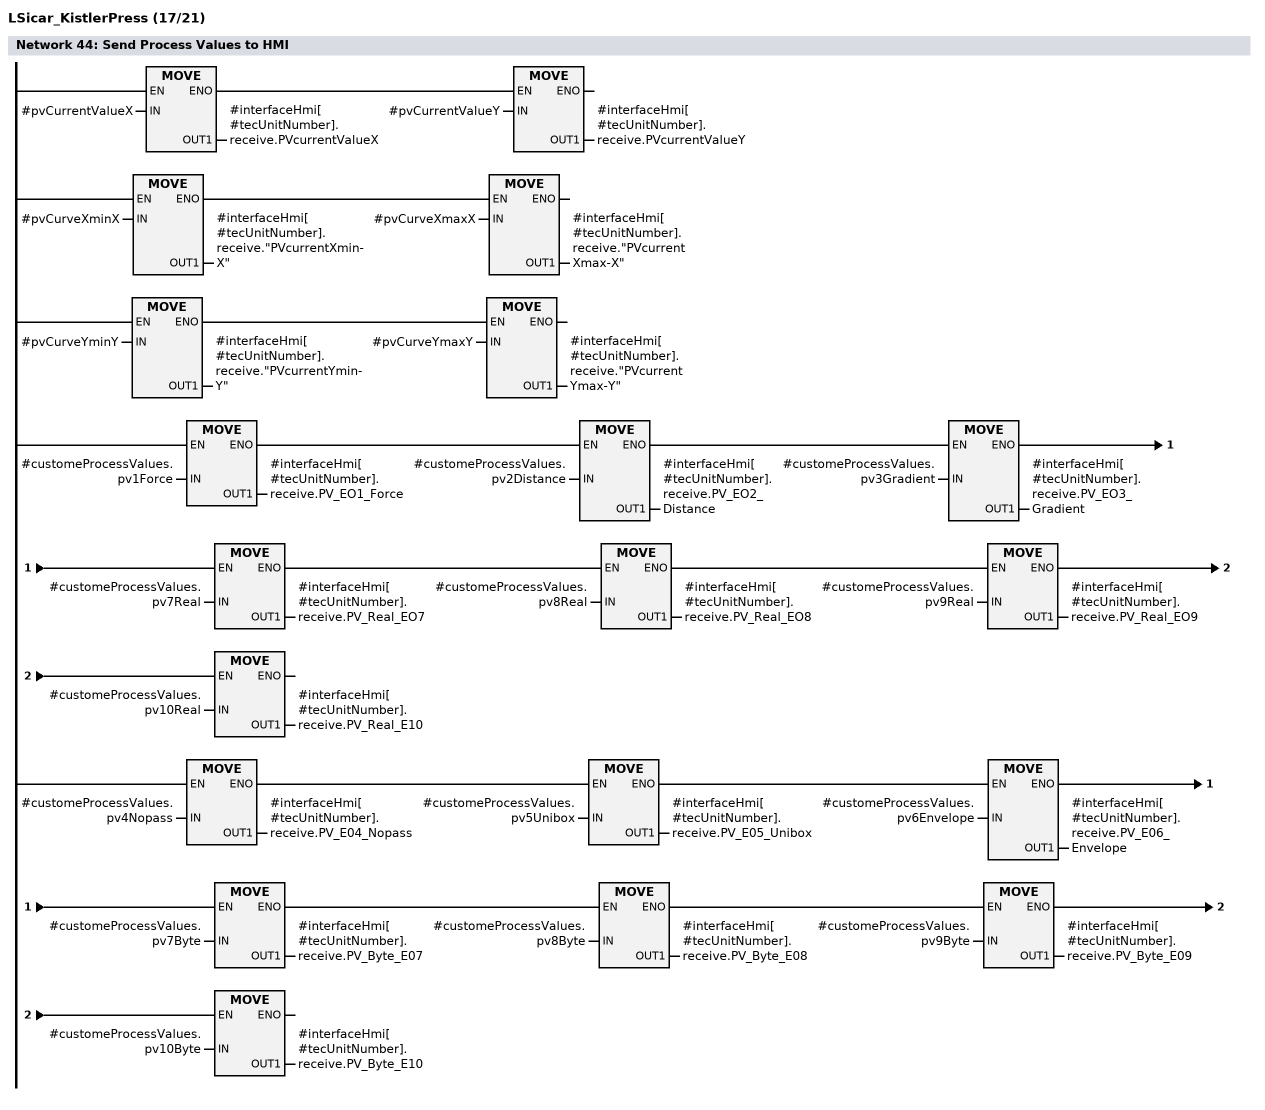
   RUNG wire#powerrail
      Move(in := #pvCurrentValueX, out1 => #interfaceHmi[#tecUnitNumber].receive.PVcurrentValueX)
      Move(in := #pvCurrentValueY, out1 => #interfaceHmi[#tecUnitNumber].receive.PVcurrentValueY)
   END_RUNG
   RUNG wire#powerrail
      Move(in := #pvCurveXminX, out1 => #interfaceHmi[#tecUnitNumber].receive."PVcurrentXmin-X")
      Move(in := #pvCurveXmaxX, out1 => #interfaceHmi[#tecUnitNumber].receive."PVcurrentXmax-X")
   END_RUNG
   RUNG wire#powerrail
      Move(in := #pvCurveYminY, out1 => #interfaceHmi[#tecUnitNumber].receive."PVcurrentYmin-Y")
      Move(in := #pvCurveYmaxY, out1 => #interfaceHmi[#tecUnitNumber].receive."PVcurrentYmax-Y")
   END_RUNG
   RUNG wire#powerrail
      Move(in := #customeProcessValues.pv1Force, out1 => #interfaceHmi[#tecUnitNumber].receive.PV_EO1_Force)
      Move(in := #customeProcessValues.pv2Distance, out1 => #interfaceHmi[#tecUnitNumber].receive.PV_EO2_Distance)
      Move(in := #customeProcessValues.pv3Gradient, out1 => #interfaceHmi[#tecUnitNumber].receive.PV_EO3_Gradient)
      Move(in := #customeProcessValues.pv7Real, out1 => #interfaceHmi[#tecUnitNumber].receive.PV_Real_EO7)
      Move(in := #customeProcessValues.pv8Real, out1 => #interfaceHmi[#tecUnitNumber].receive.PV_Real_EO8)
      Move(in := #customeProcessValues.pv9Real, out1 => #interfaceHmi[#tecUnitNumber].receive.PV_Real_EO9)
      Move(in := #customeProcessValues.pv10Real, out1 => #interfaceHmi[#tecUnitNumber].receive.PV_Real_E10)
   END_RUNG
   RUNG wire#powerrail
      Move(in := #customeProcessValues.pv4Nopass, out1 => #interfaceHmi[#tecUnitNumber].receive.PV_E04_Nopass)
      Move(in := #customeProcessValues.pv5Unibox, out1 => #interfaceHmi[#tecUnitNumber].receive.PV_E05_Unibox)
      Move(in := #customeProcessValues.pv6Envelope, out1 => #interfaceHmi[#tecUnitNumber].receive.PV_E06_Envelope)
      Move(in := #customeProcessValues.pv7Byte, out1 => #interfaceHmi[#tecUnitNumber].receive.PV_Byte_E07)
      Move(in := #customeProcessValues.pv8Byte, out1 => #interfaceHmi[#tecUnitNumber].receive.PV_Byte_E08)
      Move(in := #customeProcessValues.pv9Byte, out1 => #interfaceHmi[#tecUnitNumber].receive.PV_Byte_E09)
      Move(in := #customeProcessValues.pv10Byte, out1 => #interfaceHmi[#tecUnitNumber].receive.PV_Byte_E10)
   END_RUNG
   // the same network as SCL:
   #interfaceHmi[#tecUnitNumber].receive.PVcurrentValueX := #pvCurrentValueX;
   #interfaceHmi[#tecUnitNumber].receive.PVcurrentValueY := #pvCurrentValueY;
   #interfaceHmi[#tecUnitNumber].receive."PVcurrentXmin-X" := #pvCurveXminX;
   #interfaceHmi[#tecUnitNumber].receive."PVcurrentXmax-X" := #pvCurveXmaxX;
   #interfaceHmi[#tecUnitNumber].receive."PVcurrentYmin-Y" := #pvCurveYminY;
   #interfaceHmi[#tecUnitNumber].receive."PVcurrentYmax-Y" := #pvCurveYmaxY;
   #interfaceHmi[#tecUnitNumber].receive.PV_EO1_Force := #customeProcessValues.pv1Force;
   #interfaceHmi[#tecUnitNumber].receive.PV_EO2_Distance := #customeProcessValues.pv2Distance;
   #interfaceHmi[#tecUnitNumber].receive.PV_EO3_Gradient := #customeProcessValues.pv3Gradient;
   #interfaceHmi[#tecUnitNumber].receive.PV_Real_EO7 := #customeProcessValues.pv7Real;
   #interfaceHmi[#tecUnitNumber].receive.PV_Real_EO8 := #customeProcessValues.pv8Real;
   #interfaceHmi[#tecUnitNumber].receive.PV_Real_EO9 := #customeProcessValues.pv9Real;
   #interfaceHmi[#tecUnitNumber].receive.PV_Real_E10 := #customeProcessValues.pv10Real;
   #interfaceHmi[#tecUnitNumber].receive.PV_E04_Nopass := #customeProcessValues.pv4Nopass;
   #interfaceHmi[#tecUnitNumber].receive.PV_E05_Unibox := #customeProcessValues.pv5Unibox;
   #interfaceHmi[#tecUnitNumber].receive.PV_E06_Envelope := #customeProcessValues.pv6Envelope;
   #interfaceHmi[#tecUnitNumber].receive.PV_Byte_E07 := #customeProcessValues.pv7Byte;
   #interfaceHmi[#tecUnitNumber].receive.PV_Byte_E08 := #customeProcessValues.pv8Byte;
   #interfaceHmi[#tecUnitNumber].receive.PV_Byte_E09 := #customeProcessValues.pv9Byte;
   #interfaceHmi[#tecUnitNumber].receive.PV_Byte_E10 := #customeProcessValues.pv10Byte;
END_REGION

